									fb_ManipulatorArm( // Call Fb_Action
														(*Manipulator*)
															bCheckSensorManipulatorGripper:=GV_HMI.stTransferManipulatorToArm.bCheckSensorManipulatorGripper,
														(*Arm*)
															iGripperArmNumber:=GV_Cycle.iArmGripperLoad,
															bCheckSensorArmGripper1:=GV_HMI.stTransferManipulatorToArm.bCheckSensorArmGripper1,
															bCheckSensorArmGripper2:=GV_HMI.stTransferManipulatorToArm.bCheckSensorArmGripper2,
														(*Gripper*)
															tMouvementGripperOpen:=GV_HMI.stManipulatorGripper.tMouvementOpen,
															bCheckSensorGripperOpen:=GV_HMI.stManipulatorGripper.bCheckSensorOpen,
															tMouvementGripperClose:=GV_HMI.stManipulatorGripper.tMouvementClose,
															bCheckSensorGripperClose:=GV_HMI.stManipulatorGripper.bCheckSensorClose,
														(*Tunnel*)
															tTunnelTimeout:=GV_HMI.stManipulatorTunnel.tTimeout,
														(*Step 2_ManipulatorAboveTransfer*)
															tMove2Timeout:=T#0S, // Not used
														(*Step 3_ArmHome*)
															tMove3Timeout:=T#0S, // Not used
														(*Step 4_ManipulatorTransfer*)
															tMove4Timeout:=T#0S, // Not used
														(*Step 5_ArmTransfer*)
															tMove5Timeout:=T#0S, // Not used
														(*Step 7_ManipulatorAboveTransfer*)
															tMove7Timeout:=T#0S, // Not used
													 );
									IF fb_ManipulatorArm.bDone AND (NOT fb_ManipulatorArm.bError) THEN // Done 
										fb_ManipulatorArm.bStart:=FALSE; 
										GV_Cycle.bActionRunning:=FALSE;
										GV_Cycle.iSeqIndex:=GV_Cycle.iSeqIndex+1; 
									ELSIF fb_ManipulatorArm.bError THEN // Error
										fb_ManipulatorArm.bStart:=FALSE; 
										GV_Cycle.bActionRunning:=FALSE;
										GV_Cycle.udiErrorID:=2000+fb_ManipulatorArm.udiErrorID;
										GV_Cycle.bActionError:=TRUE;
									END_IF
									
								ENUM_Cycle_Action.ArmCNC:
								
									IF (NOT fb_ArmCNC.bInit) AND (NOT GV_Cycle.bActionRunning) THEN // Start if not already running	
										fb_ArmCNC.bStart:=TRUE;
										GV_Cycle.bActionRunning:=TRUE;
									END_IF
									
									IF fb_ArmCNC.bBusy THEN
										fb_ArmCNC.bStart:=FALSE;
									END_IF
									
									fb_ArmCNC( // Call Fb_Action
												(*TransferArmCnc*)
													bTransferArmToCnc:=GV_Cycle.bTransferArmToCnc,
													iGripperArmToCncNumber:=GV_Cycle.iGripperArmToCncNumber,
												(*TransferCncArm*)
													bTransferCncToArm:=GV_Cycle.bTransferCncToArm,
													iGripperCncToArmNumber:=GV_Cycle.iGripperCncToArmNumber,
												(*Arm*)
													bCheckSensorArmGripper1:=GV_HMI.stTransferArmCnc.bCheckSensorArmGripper1,
													bCheckSensorArmGripper2:=GV_HMI.stTransferArmCnc.bCheckSensorArmGripper2,
												(*Step 1_OpenDoor*)
													tMove1Timeout:=T#0S, // Not used
												(*Step 2_ArmInCNC*)
													tMove2Timeout:=T#0S, // Not used
												(*Step 3_WaitTransfer*)
													tMove3Timeout:=T#0S, // Not used
												(*Step 4_ArmHome*)
													tMove4Timeout:=T#0S, // Not used
												(*Step 5_CloseDoor*)
													tMove5Timeout:=T#0S, // Not used
											 );
									IF fb_ArmCNC.bDone AND (NOT fb_ArmCNC.bError) THEN // Done 
										fb_ArmCNC.bStart:=FALSE;
										GV_Cycle.bActionRunning:=FALSE; 
										GV_Cycle.iSeqIndex:=GV_Cycle.iSeqIndex+1; 
									ELSIF fb_ArmCNC.bError THEN // Error
										fb_ArmCNC.bStart:=FALSE;
										GV_Cycle.bActionRunning:=FALSE; 
										GV_Cycle.udiErrorID:=3000+fb_ArmCNC.udiErrorID;
										GV_Cycle.bActionError:=TRUE;
									END_IF
									
								ENUM_Cycle_Action.ArmToManipulator:
								
									IF (NOT fb_ArmManipulator.bInit) AND (NOT GV_Cycle.bActionRunning) THEN// Start if not already running	
										fb_ArmManipulator.bStart:=TRUE;
										GV_Cycle.bActionRunning:=TRUE;
									END_IF
									
									IF fb_ArmManipulator.bBusy THEN
										fb_ArmManipulator.bStart:=FALSE;
									END_IF
									
									fb_ArmManipulator( // Call Fb_Action
														(*Manipulator*)
															bCheckSensorManipulatorGripper:=GV_HMI.stTransferManipulatorToArm.bCheckSensorManipulatorGripper,
														(*Arm*)
															iGripperArmNumber:=GV_Cycle.iArmGripperUnload,
															bCheckSensorArmGripper1:=GV_HMI.stTransferArmToManipulator.bCheckSensorArmGripper1,
															bCheckSensorArmGripper2:=GV_HMI.stTransferArmToManipulator.bCheckSensorArmGripper2,
														(*Gripper*)
															tMouvementGripperOpen:=GV_HMI.stManipulatorGripper.tMouvementOpen,
															bCheckSensorGripperOpen:=GV_HMI.stManipulatorGripper.bCheckSensorOpen,
															tMouvementGripperClose:=GV_HMI.stManipulatorGripper.tMouvementClose,
															bCheckSensorGripperClose:=GV_HMI.stManipulatorGripper.bCheckSensorClose,
														(*Tunnel*)
															tTunnelTimeout:=GV_HMI.stManipulatorTunnel.tTimeout,
														(*Step 2_ManipulatorAboveTransfer*)
															tMove2Timeout:=T#0S, // Not used
														(*Step 3_ArmTransfer*)
															tMove3Timeout:=T#0S, // Not used
														(*Step 5_ManipulatorTransfer*)
															tMove5Timeout:=T#0S, // Not used
														(*Step 7_ArmHome*)
															tMove7Timeout:=T#0S, // Not used
														(*Step 8_ManipulatorAboveTransfer*)
															tMove8Timeout:=T#0S, // Not used
													);
									IF fb_ArmManipulator.bDone AND (NOT fb_ArmManipulator.bError) THEN // Done 
										fb_ArmManipulator.bStart:=FALSE; 
										GV_Cycle.bActionRunning:=FALSE;
										GV_Cycle.iSeqIndex:=GV_Cycle.iSeqIndex+1; 
									ELSIF fb_ArmManipulator.bError THEN // Error
										fb_ArmManipulator.bStart:=FALSE; 
										GV_Cycle.bActionRunning:=FALSE;
										GV_Cycle.udiErrorID:=4000+fb_ArmManipulator.udiErrorID;
										GV_Cycle.bActionError:=TRUE;
									END_IF
									
								ENUM_Cycle_Action.PlaceToolMagazine:
								
									IF GV_Cycle.iToolToUnloadLocationAbs=0 AND GV_Tool_Magazine.stManipulator.bToolPresenceMemory AND GV_Tool_Magazine.stManipulator.iAbsLocationNumberMemory<>GV_Cycle.iToolToLoadLocationAbs AND (NOT fb_PlaceToolMagazine.bStart) AND (NOT fb_PlaceToolMagazine.bInit) AND (NOT fb_PlaceToolMagazine.bBusy) THEN
										GV_Cycle.iToolToUnloadLocationAbs:=GV_Tool_Magazine.stManipulator.iAbsLocationNumberMemory;
									END_IF

									IF GV_Cycle.iToolToUnloadLocationAbs>0 THEN	
										//ICI -> Vérifier que emplacement disponible ? mémoire emplacement ou faire la vérif, avec outil en pince possible ?

										IF (NOT fb_PlaceToolMagazine.bInit) AND (NOT GV_Cycle.bActionRunning) THEN // Start if not already running		
											fb_PlaceToolMagazine.bStart:=TRUE;
											GV_Cycle.bActionRunning:=TRUE;
										END_IF
										
										IF fb_PlaceToolMagazine.bBusy THEN
											fb_PlaceToolMagazine.bStart:=FALSE;
										END_IF
										
										fb_PlaceToolMagazine( // Call Fb_Action
															(*ToolLocation*)
																stToolLocation:=GV_Tool_Magazine.aLocation[GV_Cycle.iToolToUnloadLocationAbs],
																lrZToolOffset:=GV_Tool_Magazine.lrZOffsetAboveLocation,//17.5,
															(*Manipulator*)
																bCheckSensorManipulatorGripper:=GV_HMI.stPickToolMagazine.bCheckSensorManipulatorGripper,
															(*Gripper*)
																tMouvementGripperOpen:=GV_HMI.stManipulatorGripper.tMouvementOpen,
																bCheckSensorGripperOpen:=GV_HMI.stManipulatorGripper.bCheckSensorOpen,
																tMouvementGripperClose:=GV_HMI.stManipulatorGripper.tMouvementClose,
																bCheckSensorGripperClose:=GV_HMI.stManipulatorGripper.bCheckSensorClose,
															(*Tunnel*)
																tTunnelTimeout:=GV_HMI.stManipulatorTunnel.tTimeout,
															(*Breakage*)
																tBreakageTimeout:=GV_HMI.stManipulatorBreakage.tTimeout,
																lrBreakageZOffsetSensor:=GV_HMI.stManipulatorBreakage.lrOffsetSensor,
																lrBreakageToleranceLength:=GV_HMI.stManipulatorBreakage.lrToleranceLength,
																lrBreakageVelocity:=GV_HMI.stManipulatorBreakage.lrMeasureVelocity,
															(*Step 4_FrontLocation*)
																tMove4Timeout:=T#0S, // Not used
															(*Step 6_AboveLocation*)
																tMove6Timeout:=T#0S, // Not used
															(*Step 8_FrontLocation*)
																tMove8Timeout:=T#0S, // Not used
															);
										IF fb_PlaceToolMagazine.bDone AND (NOT fb_PlaceToolMagazine.bError) THEN // Done 
											fb_PlaceToolMagazine.bStart:=FALSE; 
											GV_Cycle.bActionRunning:=FALSE;
											GV_Cycle.iToolToUnloadLocationAbs:=0;
											GV_Cycle.iSeqIndex:=GV_Cycle.iSeqIndex+1; 
										ELSIF fb_PlaceToolMagazine.bError THEN // Error
											GV_Cycle.udiErrorID:=5000+fb_PlaceToolMagazine.udiErrorID;
											GV_Cycle.bActionError:=TRUE;
										END_IF
										
									ELSE
										GV_Cycle.iSeqIndex:=GV_Cycle.iSeqIndex+1;
									END_IF
	
							END_CASE
							
						(* Action Error *)
							IF GV_Cycle.bActionError THEN // Action in Error
								(*Log*)
									PRG_Log_WM.fbLogWM.M_Write_Log('Cycle Step : 5_ExecuteSequence=Error');
									PRG_Log_WM.fbLogWM.M_Write_Log(CONCAT('Cycle Step : ErrorID=',UDINT_TO_STRING(GV_Cycle.udiErrorID)));
								GV_Cycle.eCycleStep:=ENUM_Cycle_Step.Error; // Go to Step Error
							END_IF		
				
					ELSE
						bExecuteSequenceDone:=TRUE;
					END_IF
					
				(* Next Step *)	
					IF bExecuteSequenceDone THEN
						GV_Cycle.eCycleStep:=ENUM_Cycle_Step.End; // Go to Step End
					END_IF
				
			ENUM_Cycle_Step.End: // Step End = 7
				bEndDone:=FALSE;
				GV_Cycle.iToolToUnloadLocationAbs:=0;
				(* End *)
					// ...
					IF ((GV_Cycle.bStartStop AND GV_Axes.bAxisAllNotMoving)
					OR ((NOT GV_Cycle.bStartStop) AND GV_Axes.stAxisX.bHaltDone AND GV_Axes.stAxisY.bHaltDone AND GV_Axes.stAxisZ.bHaltDone AND GV_Axes.stAxisArm.bHaltDone AND GV_Axes.bAxisAllNotMoving)) THEN
						GV_Axes.stAxisX.bAutoCmdAbs:=FALSE;
						GV_Axes.stAxisY.bAutoCmdAbs:=FALSE;
						GV_Axes.stAxisZ.bAutoCmdAbs:=FALSE;
						GV_Axes.stAxisArm.bAutoCmdAbs:=FALSE;
						bEndDone:=TRUE;
					END_IF

					//IF ((NOT GV_Cycle.bStartStop) AND GV_Axes.stAxisX.bStopDone AND GV_Axes.stAxisY.bStopDone AND GV_Axes.stAxisZ.bStopDone AND GV_Axes.stAxisArm.bStopDone AND GV_Axes.bAxisAllNotMoving) THEN
					//	bEndDone:=TRUE;
					//END_IF
					
				(* Next Step *)	
					IF bEndDone THEN
						GV_Cycle.eCycleStep:=ENUM_Cycle_Step.InitData; // Go to Step InitData
					END_IF
	
			ENUM_Cycle_Step.Error: // Step Error = 9
				bErrorDone:=FALSE;
				GV_Cycle.iToolToUnloadLocationAbs:=0;
				(* Error *)
					// ...
					GV_Axes.stAxisX.bAutoCmdAbs:=FALSE;
					GV_Axes.stAxisY.bAutoCmdAbs:=FALSE;
					GV_Axes.stAxisZ.bAutoCmdAbs:=FALSE;
					GV_Axes.stAxisArm.bAutoCmdAbs:=FALSE;
					
					GV_Cycle.bStartStop:=FALSE;
					GV_Cycle.bInitCycleDone:=FALSE;
					
					IF GV_Cycle.bResetError THEN
						bErrorDone:=TRUE;
					END_IF
				(* Next Step *)	
					IF bErrorDone THEN
						GV_Cycle.bActionRunning:=FALSE;
						GV_Cycle.bActionError:=FALSE;
						GV_Cycle.udiErrorID:=0;
						GV_Cycle.eCycleStep:=ENUM_Cycle_Step.InitData;
					END_IF
			
		END_CASE
		
	END_IF

(** CYCLE IN PROGRESS **)
GV_Cycle.bCycleInProgress:=GV_Cycle.eCycleStep<>ENUM_Cycle_Step.InitAll AND GV_Cycle.eCycleStep<>ENUM_Cycle_Step.InitData;

(** LOG CYCLE STEP **)
	(* Text CycleStep *)
		CASE GV_Cycle.eCycleStep OF
				ENUM_Cycle_Step.InitAll:           	sTxtCycleStep:='0_InitAll';
				ENUM_Cycle_Step.InitData:           sTxtCycleStep:='0_InitData';
				ENUM_Cycle_Step.Ready:          	sTxtCycleStep:='2_Ready';
				ENUM_Cycle_Step.Preparation:        sTxtCycleStep:='3_Preparation';
				ENUM_Cycle_Step.BuildSequence:  	sTxtCycleStep:='4_BuildSequence';
				ENUM_Cycle_Step.ExecuteSequence:	sTxtCycleStep:='5_ExecuteSequence';
				ENUM_Cycle_Step.End:            	sTxtCycleStep:='7_End';
				ENUM_Cycle_Step.Abort:          	sTxtCycleStep:='8_Abort';
				ENUM_Cycle_Step.Error:         		sTxtCycleStep:='9_Error';
		END_CASE
	(* Text CyclePrevStep *)
		CASE GV_Cycle.eCyclePrevStep OF
				ENUM_Cycle_Step.InitAll:           	sTxtCycleStep:='0_InitAll';
				ENUM_Cycle_Step.InitData:           sTxtCycleStep:='0_InitData';
				ENUM_Cycle_Step.Ready:          	sTxtCycleStep:='2_Ready';
				ENUM_Cycle_Step.Preparation:        sTxtCycleStep:='3_Preparation';
				ENUM_Cycle_Step.BuildSequence:  	sTxtCycleStep:='4_BuildSequence';
				ENUM_Cycle_Step.ExecuteSequence:	sTxtCycleStep:='5_ExecuteSequence';
				ENUM_Cycle_Step.End:            	sTxtCycleStep:='7_End';
				ENUM_Cycle_Step.Abort:          	sTxtCycleStep:='8_Abort';
				ENUM_Cycle_Step.Error:         		sTxtCycleStep:='9_Error';
		END_CASE
	(* Log *)
		sTextLog:=(CONCAT('Cycle Step ',CONCAT(sTxtCyclePrevStep,CONCAT('-> ',sTxtCycleStep))));	
		IF GV_OpMode.eOpMode=ENUM_OpMode.AUTO AND GV_Cycle.eCycleStep<>GV_Cycle.eCyclePrevStep THEN
			PRG_Log_WM.fbLogWM.M_Write_Log(sTextLog);
			GV_Cycle.eCyclePrevStep:=GV_Cycle.eCycleStep; // Previous Step := Step in progress
		END_IF

END_PROGRAM

// ---- 08_Cycle/03_POUs/02_FBs/FB_20_Action_Initialization.TcPOU
FUNCTION_BLOCK FB_20_Action_Initialization
VAR_INPUT
	(** SETUP ST **)
		//stToolLocation : ST_Tool_Location ; // Tool_Location structure of the Tool to Pick
		
	(** SETUP TIME **)
		(*Manipulator Gripper mvmnt*)
			//tMouvementGripperOpen : TIME ; // Value of the manipulator gripper open mouvement duration
			//tMouvementGripperClose : TIME ; // Value of the manipulator gripper close mouvement duration
		(*Tunnel*)
			tTunnelTimeout : TIME ; // Value of the timeout for travel the tunnel
		(*Step 2*)
			tMove2Timeout : TIME ; // Value of the timeout for Step 2

	(** SETUP FLAG **)
		//bCheckSensorManipulatorGripper : BOOL ; // Check the manipulator gripper sensor at the beginning
		(*Gripper*)
			//bCheckSensorGripperOpen : BOOL ; // Check the manipulator gripper sensor after open
			//bCheckSensorGripperClose : BOOL ; // Check the manipulator gripper sensor after close	
			
	(** PROCESS FLAG **)
	    bInit : BOOL ; // Init the Fb
	    bStart : BOOL ; // Start the Fb
END_VAR
VAR_OUTPUT
	(** PROCESS UDINT **)
		udiErrorID : UDINT ; // Fb Error ID
		
	(** PROCESS FLAG **)
		bBusy  : BOOL ; // Fb is Busy
		bDone  : BOOL ; // Fb is Done
		bError : BOOL ; // Fb in Error
END_VAR
VAR_IN_OUT
END_VAR	
VAR
	(** SETUP ENUM **)
		(*Manipulator Gripper mvmnt*)
			//eGripperMode : ENUM_Gripper_Mode; // Gripper mode for gripper mouvement (fbGripper)
		(*Tunnel*)
			eTunnelMode : ENUM_Tunnel_Mode; // Tunnel mode for travel (fbTunnel)

	(** SETUP TIME **)
		(*Manipulator Gripper mvmnt*)
			//tGripperTime : TIME ; // Mouvement duration for gripper mouvement (fbGripper)
	
	(** SETUP FLAG **)
		(*Manipulator Gripper mvmnt*)
			//bGripperSensor : BOOL ; // Sensor check for gripper mouvement (fbGripper)
		
	(** PROCESS STRING **)
		strTextLog : STRING ; // Text to Log
		
	(** PROCESS LREAL **)
		
	(** PROCESS INT **)
		iStep  : INT := 0 ; // Step of the Fb
		iSubStep : INT := 0 ; // SubStep of the Fb
		iPrevStep : INT := 0 ; // Previous Step of the Fb
		iPrevSubStep : INT := 0 ; // Previous Subtep of the Fb
		
	(** PROCESS FLAG + R_TRIG **)
		rtInit : R_TRIG ; // FB Init at rising edge
		rtStart : R_TRIG ; // FB Start at rising edge
		(*Tunnel*)
			bTunnelTravel : BOOL ; // Need to travel the tunnel
		bXError : BOOL ; // Axis X Error
		bYError : BOOL ; // Axis Y Error
		bZError : BOOL ; // Axis Z Error
		bArmError : BOOL ; // Axis Arm Error
	
	(** FB **)
		(*Gripper*)
			//fbGripper : FB_Manipulator_Gripper ;
		(*Tunnel*)
			fbTunnel : FB_Manipulator_Tunnel ;
		(*Step 2*)
			tonTimeoutMove2 : TON ; // TON timeout for the Step 2
END_VAR

//-----------------------------------------------------------------------------------------
//
//                  			FB_20_Action_Initialization
//
//						Management of the Initialization process
//-----------------------------------------------------------------------------------------
//
//Auteur: G.GOETZ
//Création: 13.03.2026
//Dernière modification : 13.03.2026 (G.GOETZ)
//       			
//-----------------------------------------------------------------------------------------
//
//     							Liste des modifications  	
//
// 13.03.2026 (G.GOETZ) -> Création		
//-----------------------------------------------------------------------------------------

(** FB CALL **)
	rtInit(CLK:=bInit);
	rtStart(CLK:=bStart);
	fbTunnel( // Call Tunnel travel
			eTunnelMode:=eTunnelMode,
			tTimeout:=tTunnelTimeout
			);

(** AXIS ERRORS **)
	bXError:=(GV_Axes.stAxisX.stDriveAx8206.AxisRef.Status.Error OR GV_Axes.stAxisX.stDriveAx8206.AxisRef.Status.ErrorStop OR GV_Axes.stAxisX.stDriveAx8206.AxisRef.Status.ErrorID<>0);
	bYError:=(GV_Axes.stAxisY.stDriveAx8206.AxisRef.Status.Error OR GV_Axes.stAxisY.stDriveAx8206.AxisRef.Status.ErrorStop OR GV_Axes.stAxisY.stDriveAx8206.AxisRef.Status.ErrorID<>0);
	bZError:=(GV_Axes.stAxisZ.stDriveAx8206.AxisRef.Status.Error OR GV_Axes.stAxisZ.stDriveAx8206.AxisRef.Status.ErrorStop OR GV_Axes.stAxisZ.stDriveAx8206.AxisRef.Status.ErrorID<>0);
	bArmError:=(GV_Axes.stAxisArm.stDriveAx8206.AxisRef.Status.Error OR GV_Axes.stAxisArm.stDriveAx8206.AxisRef.Status.ErrorStop OR GV_Axes.stAxisArm.stDriveAx8206.AxisRef.Status.ErrorID<>0);


(** INIT **)
	IF (rtinit.Q OR bInit) AND (NOT bStart) THEN
		bBusy:=FALSE;
		bDone:=FALSE;
		bError:=FALSE;
		udiErrorID:=0;
		iStep:=0;
		iSubStep:=0;
		bInit:=FALSE;
	END_IF

(** STEPS **)
    CASE iStep OF
		
        0: (* Step 0 = Idle + Check *)
            bBusy:=FALSE;
            bDone:=FALSE;
			bError:=FALSE;
			udiErrorID:=0;
			iSubStep:=0;
			
			tonTimeoutMove2.IN:=FALSE;
			//tonTimeoutMove4.IN:=FALSE;
			//tonTimeoutMove6.IN:=FALSE;
			//tonTimeoutMove8.IN:=FALSE;
			
			GV_Axes.stAxisX.bAutoCmdAbs:=FALSE;
			GV_Axes.stAxisY.bAutoCmdAbs:=FALSE;
			GV_Axes.stAxisZ.bAutoCmdAbs:=FALSE;
			GV_Axes.stAxisArm.bAutoCmdAbs:=FALSE;
			
			fbTunnel.bInit:=TRUE;
			
			bTunnelTravel:=FALSE;

			(* Idle->Start *)
				IF rtStart.Q AND (NOT bInit) THEN
					bBusy:=TRUE;
					(*Log*)
						PRG_Log_WM.fbLogWM.M_Write_Log('FB_20_Action_Initialization : 0_Idle : Init of the Magazine');
						//IF Exemple THEN
						//	strTextLog:='With';
						//ELSE
						//	strTextLog:='Without';
						//END_IF
						//PRG_Log_WM.fbLogWM.M_Write_Log(CONCAT('FB_20_Action_Initialization : 0_Idle : Exemple Check = ',strTextLog));
							
					(* Check xxx *)

					IF (NOT bError) THEN
						(*Log*)
							PRG_Log_WM.fbLogWM.M_Write_Log('FB_20_Action_Initialization : 0_Idle->1_Tunnel');
						iStep:=1; // Next Step
					END_IF

				END_IF
	
		1: (* Step 1 = Tunnel passage (if needed) *)
			IF (NOT bTunnelTravel) THEN
				IF GV_Tool_Magazine.stManipulator.ePositionMag=ENUM_Position_Magazine.Top THEN
					bTunnelTravel:=FALSE;
					(*Log*)
						PRG_Log_WM.fbLogWM.M_Write_Log('FB_20_Action_Initialization : 1_Tunnel : No Need to Travel');
						PRG_Log_WM.fbLogWM.M_Write_Log('FB_20_Action_Initialization : 1_Tunnel->2_???');
					iStep:=2; // Next Step
				END_IF	
				IF GV_Tool_Magazine.stManipulator.ePositionMag=ENUM_Position_Magazine.Bottom THEN
					eTunnelMode:=ENUM_Tunnel_MODE.BottomToTop;
					bTunnelTravel:=TRUE;
					(*Log*)
						PRG_Log_WM.fbLogWM.M_Write_Log('FB_20_Action_Initialization : 1_Tunnel : Need to Travel Bottom->Top');
				END_IF			
				IF GV_Tool_Magazine.stManipulator.ePositionMag=ENUM_Position_Magazine.Unknow THEN // Manipulator Unknow position
					bError:=TRUE;
					udiErrorID:=101; // 101 = Step 1 Error Tunnel 01
					fbTunnel.bStart:=FALSE;
					bTunnelTravel:=FALSE;
					(*Log*)
						PRG_Log_WM.fbLogWM.M_Write_Log('FB_20_Action_Initialization : 1_Tunnel=Error');
						PRG_Log_WM.fbLogWM.M_Write_Log(CONCAT('FB_20_Action_Initialization : ErrorID=',UDINT_TO_STRING(udiErrorID)));
					iStep:=0; // Idle Step
				END_IF
			END_IF
			
			IF bTunnelTravel AND (NOT fbTunnel.bStart) AND (NOT fbTunnel.bBusy) THEN // Tunnel Start
				fbTunnel.bStart:=TRUE;
			END_IF
			IF fbTunnel.bDone THEN // Tunnel Done
				fbTunnel.bStart:=FALSE;
				bTunnelTravel:=FALSE;
				(*Log*)
					PRG_Log_WM.fbLogWM.M_Write_Log('FB_20_Action_Initialization : 1_Tunnel->2_???');
				iStep:=2; // Next Step
			ELSIF fbTunnel.bError THEN // Tunnel Error
				bError:=TRUE;
				udiErrorID:=100+fbTunnel.udiErrorID; // 1xx = Step 1 Error + Error xx fbTunnel
				fbTunnel.bStart:=FALSE;
				bTunnelTravel:=FALSE;
				(*Log*)
					PRG_Log_WM.fbLogWM.M_Write_Log('FB_20_Action_Initialization : 1_Tunnel=Error');
					PRG_Log_WM.fbLogWM.M_Write_Log(CONCAT('FB_20_Action_Initialization : ErrorID=',UDINT_TO_STRING(udiErrorID)));
				iStep:=0; // Idle Step
			END_IF
		
		2: (* Step 2 = Move the manipulator to Home (Y->Z->X) *)
			tonTimeoutMove2.PT:=tMove2Timeout;
			tonTimeoutMove2.IN:=TRUE;
			
			CASE iSubStep OF
        
				0: (* Start Y move *)
					GV_Axes.stAxisY.lrAutoPosAbs:=GV_Tool_Magazine.stManipulator.lrYHome;
					GV_Axes.stAxisY.bAutoCmdAbs:=TRUE;
					(*Log*)
						PRG_Log_WM.fbLogWM.M_Write_Log('FB_20_Action_Initialization : 2_MoveHome : 0 : Start Y move');
					iSubStep:=1; // Next SubStep

				1: (* Wait Y move done *)
				   IF GV_Axes.stAxisY.bAutoDone AND (NOT bYError) THEN
						GV_Axes.stAxisY.bAutoCmdAbs:=FALSE;
						(*Log*)
							PRG_Log_WM.fbLogWM.M_Write_Log('FB_20_Action_Initialization : 2_MoveHome : 1 : Y move done');
						iSubStep:=2; // Next SubStep
					ELSIF bYError THEN
						bError:=TRUE;
						udiErrorID:=211; // 211 = Step 2 SubStep 1 Error Axis Y 1
						GV_Axes.stAxisY.bAutoCmdAbs:=FALSE;
						tonTimeoutMove2.IN:=FALSE;
						(*Log*)
							PRG_Log_WM.fbLogWM.M_Write_Log('FB_20_Action_Initialization : 2_MoveHome=Error');
							PRG_Log_WM.fbLogWM.M_Write_Log(CONCAT('FB_20_Action_Initialization : ErrorID=',UDINT_TO_STRING(udiErrorID)));
						iSubStep:=0; // Stop SubStep
						iStep:=0; // Idle Step
					END_IF
				
				2: (* Start Z move *)
					GV_Axes.stAxisZ.lrAutoPosAbs:=GV_Tool_Magazine.stManipulator.lrZHome;
					GV_Axes.stAxisZ.bAutoCmdAbs:=TRUE;
					(*Log*)
						PRG_Log_WM.fbLogWM.M_Write_Log('FB_20_Action_Initialization : 2_MoveHome : 2 : Start Z move');
					iSubStep:=3; // Next SubStep

				3: (* Wait Z move done *)
				   IF GV_Axes.stAxisZ.bAutoDone AND (NOT bZError) THEN
						GV_Axes.stAxisZ.bAutoCmdAbs:=FALSE;
						(*Log*)
							PRG_Log_WM.fbLogWM.M_Write_Log('FB_20_Action_Initialization : 2_MoveHome : 3 : Z move done');
						iSubStep:=4; // Next SubStep
					ELSIF bZError THEN
						bError:=TRUE;
						udiErrorID:=231; // 231 = Step 2 SubStep 3 Error Axis Z 1
						GV_Axes.stAxisZ.bAutoCmdAbs:=FALSE;
						tonTimeoutMove2.IN:=FALSE;
						(*Log*)
							PRG_Log_WM.fbLogWM.M_Write_Log('FB_20_Action_Initialization : 2_MoveHome=Error');
							PRG_Log_WM.fbLogWM.M_Write_Log(CONCAT('FB_20_Action_Initialization : ErrorID=',UDINT_TO_STRING(udiErrorID)));
						iSubStep:=0; // Stop SubStep
						iStep:=0; // Idle Step
					END_IF

				4: (* Start X move *)
					GV_Axes.stAxisX.lrAutoPosAbs:=GV_Tool_Magazine.stManipulator.lrXHome;
					GV_Axes.stAxisX.bAutoCmdAbs:=TRUE;
					(*Log*)
						PRG_Log_WM.fbLogWM.M_Write_Log('FB_20_Action_Initialization : 2_MoveHome : 4 : Start X move');
					iSubStep:=5; // Next Step

				5: (* Wait X move done *)
				   IF GV_Axes.stAxisX.bAutoDone AND (NOT bXError) THEN
						GV_Axes.stAxisX.bAutoCmdAbs:=FALSE;
						tonTimeoutMove2.IN:=FALSE;
						(*Log*)
							PRG_Log_WM.fbLogWM.M_Write_Log('FB_20_Action_Initialization : 2_MoveHome : 5 : X move done');
							PRG_Log_WM.fbLogWM.M_Write_Log('FB_20_Action_Initialization : 2_MoveHome->0_Idle');
						iSubStep:=0; // End SubStep
						iStep:=0; // End Step
						bDone:=TRUE;
						bBusy:=FALSE;
					ELSIF bXError THEN
						bError:=TRUE;
						udiErrorID:=251; // 251 = Step 2 SubStep 5 Error Axis X 1
						GV_Axes.stAxisX.bAutoCmdAbs:=FALSE;
						tonTimeoutMove2.IN:=FALSE;
						(*Log*)
							PRG_Log_WM.fbLogWM.M_Write_Log('FB_20_Action_Initialization : 2_MoveHome=Error');
							PRG_Log_WM.fbLogWM.M_Write_Log(CONCAT('FB_20_Action_Initialization : ErrorID=',UDINT_TO_STRING(udiErrorID)));
						iSubStep:=0; // Stop SubStep
						iStep:=0; // Idle Step
					END_IF
					
			END_CASE	
		
			IF tonTimeoutMove2.Q AND tonTimeoutMove2.PT<>T#0S THEN // Timeout 
				bError:=TRUE;
				udiErrorID:=299; // 299 = Step 2 Error Timeout 99
				GV_Axes.stAxisZ.bAutoCmdAbs:=FALSE;
				GV_Axes.stAxisX.bAutoCmdAbs:=FALSE;
				GV_Axes.stAxisY.bAutoCmdAbs:=FALSE;
				tonTimeoutMove2.IN:=FALSE;
				(*Log*)
					PRG_Log_WM.fbLogWM.M_Write_Log('FB_20_Action_Initialization : 2_MoveHome=Error');
					PRG_Log_WM.fbLogWM.M_Write_Log(CONCAT('FB_20_Action_Initialization : ErrorID=',UDINT_TO_STRING(udiErrorID)));
				iSubStep:=0;
				iStep:=0;
			END_IF
			
			
			
			
	END_CASE

END_FUNCTION_BLOCK

// ---- 09_Tool_Magazine/03_POUs/02_FBs/FB_Manipulator_Tunnel.TcPOU
FUNCTION_BLOCK FB_Manipulator_Tunnel
VAR_INPUT
	(** SETUP ENUM **)
		eTunnelMode : ENUM_Tunnel_Mode ; // Mode of the tunnel	

	(** SETUP TIME **)
		tTimeout : TIME ; // Max time for travel the tunnel

	(** PROCESS FLAG **)
		bInit : BOOL ; // Init the FB
	    bStart : BOOL ; // Start the Fb
END_VAR
VAR_OUTPUT
	(** PROCESS UDINT **)
		udiErrorID : UDINT ; // Fb Error ID
		
	(** PROCESS FLAG **)
		bBusy  : BOOL ; // Fb is Busy
		bDone  : BOOL ; // Fb is Done
		bError : BOOL ; // Fb in Error
END_VAR
VAR_IN_OUT
END_VAR	
VAR
	(** STRING **)
		strTextLog : STRING ; // Text to Log

	(** PROCESS INT **)
		iStep  : INT := 0 ; // Step of the Fb
		iSubStep : INT := 0 ; // SubStep of the Fb
		iPrevStep : INT := 0 ; // Previous Step of the Fb
		iPrevSubStep : INT := 0 ; // Previous Subtep of the Fb
	
	(** PROCESS FLAG + R_TRIG **)
		rtInit : R_TRIG ; // FB Init at rising edge
		rtStart : R_TRIG ; // FB Start at rising edge
		bTunnelTravelDone : BOOL ; // Tunnel travel done
		bXError : BOOL ; // Axis X Error
		bYError : BOOL ; // Axis Y Error
		bZError : BOOL ; // Axis Z Error
		bArmError : BOOL ; // Axis Arm Error
		
	(** FB **)
		tonTimeout : TON ; // TON timeout of the tunnel travel
END_VAR

//-----------------------------------------------------------------------------------------
//
//                  		FB_Manipulator_Tunnel
//
//			Management of the manipulator passage through the tunnel
//-----------------------------------------------------------------------------------------
//
//Auteur: G.GOETZ
//Création: 06.02.2026
//Dernière modification : 08.04.2026 (G.GOETZ)
//       			
//-----------------------------------------------------------------------------------------
//
//     							Liste des modifications  	
//
// 06.02.2026 (G.GOETZ) -> Création
// 08.04.2026 (G.GOETZ) -> Ajout Init + Modification du cycle
//-----------------------------------------------------------------------------------------

(** FB CALL **)
	rtInit(CLK:=bInit);
	rtStart(CLK:=bStart);
	
	tonTimeout();

(** AXIS ERRORS **)
	bXError:=(GV_Axes.stAxisX.stDriveAx8206.AxisRef.Status.Error OR GV_Axes.stAxisX.stDriveAx8206.AxisRef.Status.ErrorStop OR GV_Axes.stAxisX.stDriveAx8206.AxisRef.Status.ErrorID<>0);
	bYError:=(GV_Axes.stAxisY.stDriveAx8206.AxisRef.Status.Error OR GV_Axes.stAxisY.stDriveAx8206.AxisRef.Status.ErrorStop OR GV_Axes.stAxisY.stDriveAx8206.AxisRef.Status.ErrorID<>0);
	bZError:=(GV_Axes.stAxisZ.stDriveAx8206.AxisRef.Status.Error OR GV_Axes.stAxisZ.stDriveAx8206.AxisRef.Status.ErrorStop OR GV_Axes.stAxisZ.stDriveAx8206.AxisRef.Status.ErrorID<>0);
	bArmError:=(GV_Axes.stAxisArm.stDriveAx8206.AxisRef.Status.Error OR GV_Axes.stAxisArm.stDriveAx8206.AxisRef.Status.ErrorStop OR GV_Axes.stAxisArm.stDriveAx8206.AxisRef.Status.ErrorID<>0);

(** INIT **)
	IF (rtinit.Q OR bInit) AND (NOT bStart) THEN
		iStep:=0;
		bInit:=FALSE;
	END_IF

(** STEPS **)
    CASE iStep OF
		
        0: (* Step 0 = Idle *)
            bBusy:=FALSE;
            bDone:=FALSE;
			bError:=FALSE;
			udiErrorID:=0;
			iSubStep:=0;
			
			tonTimeout.IN:=FALSE;
			
			bTunnelTravelDone:=FALSE;
			
			(* Idle->Setup *)
				IF bStart AND (NOT bInit) THEN
					bBusy:=TRUE;
					(*Log*)
						PRG_Log_WM.fbLogWM.M_Write_Log('FB_Manipulator_Tunnel : 0_Idle->1_Setup');
					iStep:=1; // Next Step
				END_IF
				
		1: (* Step 1 = Setup *)
			(*Log*)
				(*TunnelMode*)
					CASE eTunnelMode OF
						ENUM_Tunnel_Mode.TopToBottom:		strTextLog:='TopToBottom';
						ENUM_Tunnel_Mode.BottomToTop:		strTextLog:='BottomToTop';
					END_CASE
					PRG_Log_WM.fbLogWM.M_Write_Log(CONCAT('FB_Manipulator_Tunnel : 1_Setup : Tunnel Mode = ',strTextLog));
				(*Timeout*)
					strTextLog:=TIME_TO_STRING(tTimeout);
					PRG_Log_WM.fbLogWM.M_Write_Log(CONCAT('FB_Manipulator_Tunnel : 1_Setup : Timeout = ',strTextLog));				
				PRG_Log_WM.fbLogWM.M_Write_Log('FB_Manipulator_Tunnel : 1_Setup->2_Process');
				
			tonTimeout.PT:=tTimeout;
			iStep:=2; // Next Step
			
		2: (* Step 2 = Process (Y->(ZLowestRacKTop)->(XFirst)) *)
			tonTimeout.IN:=TRUE; // Start TON timeout

				CASE iSubStep OF
		
					0: (* Start Y move *)
						GV_Axes.stAxisY.lrAutoPosAbs:=GV_Tool_Magazine.stManipulator.lrYTunnel;
						GV_Axes.stAxisY.bAutoCmdAbs:=TRUE;
						(*Log*)
							PRG_Log_WM.fbLogWM.M_Write_Log('FB_Manipulator_Tunnel : 2_Process : 0 : Start Y move');
						iSubStep:=1; // Next SubStep
						
					1: (* Wait Y move done *)
					   IF GV_Axes.stAxisY.bAutoDone AND (NOT bYError) THEN
							GV_Axes.stAxisY.bAutoCmdAbs:=FALSE;
							(*Log*)
								PRG_Log_WM.fbLogWM.M_Write_Log('FB_Manipulator_Tunnel : 2_Process : 1 : Y move done');

							CASE eTunnelMode OF 
								ENUM_Tunnel_Mode.TopToBottom: // X Top
									IF GV_Tool_Magazine.stManipulator.lrZPosition<GV_Tool_Magazine.lrZLowestRackTop+40 THEN
										(*Log*)
											PRG_Log_WM.fbLogWM.M_Write_Log('FB_Manipulator_Tunnel : 2_Process : 1->2 : ZLowestRackTop');
										iSubStep:=2; // Next SubStep
									ELSE
										IF GV_Tool_Magazine.stManipulator.lrXPosition<GV_Tool_Magazine.lrXFirstLocationTop THEN
											(*Log*)
												PRG_Log_WM.fbLogWM.M_Write_Log('FB_Manipulator_Tunnel : 2_Process : 1->4 : XFirstTop');
											iSubStep:=4; // Next SubStep
										ELSE
											(*Log*)
												PRG_Log_WM.fbLogWM.M_Write_Log('FB_Manipulator_Tunnel : 2_Process -> 3_Process');
											iSubStep:=0; // End SubStep
											iStep:=3; // Next Stpe
										END_IF
									END_IF
								ENUM_Tunnel_Mode.BottomToTop: // X Bottom
									IF GV_Tool_Magazine.stManipulator.lrXPosition<GV_Tool_Magazine.lrXFirstLocationBottom+GV_Tool_Magazine.lrXLocationOffsetBottom THEN
										(*Log*)
											PRG_Log_WM.fbLogWM.M_Write_Log('FB_Manipulator_Tunnel : 2_Process : 1->4 : XFirstBottom');
										iSubStep:=4; // Next SubStep
									ELSE
										(*Log*)
											PRG_Log_WM.fbLogWM.M_Write_Log('FB_Manipulator_Tunnel : 2_Process -> 3_Process');
											iSubStep:=0; // End SubStep
											iStep:=3; // Next Stpe
									END_IF
							END_CASE
						ELSIF bYError THEN
							bError:=TRUE;
							udiErrorID:=21; // 21 = Step 2 SubStep 1 Error Axis Y
							GV_Axes.stAxisY.bAutoCmdAbs:=FALSE;
							tonTimeout.IN:=FALSE;
							(*Log*)
								PRG_Log_WM.fbLogWM.M_Write_Log('FB_Manipulator_Tunnel : 2_Process=Error');
								PRG_Log_WM.fbLogWM.M_Write_Log(CONCAT('FB_Manipulator_Tunnel : ErrorID=',UDINT_TO_STRING(udiErrorID)));
							iSubStep:=0; // Stop SubStep
							iStep:=0; // Idle Step
						END_IF

					2: (* Start ZLowestRackTop move *)
						GV_Axes.stAxisZ.lrAutoPosAbs:=GV_Tool_Magazine.lrZLowestRackTop+40;
						(*Log*)
							PRG_Log_WM.fbLogWM.M_Write_Log('FB_Manipulator_Tunnel : 2_Process : 2 : Start ZLowestRackTop move');
						GV_Axes.stAxisZ.bAutoCmdAbs:=TRUE;
						iSubStep:=3; // Next SubStep

					3: (* Wait ZLowestRackTop move done *)
					   IF GV_Axes.stAxisZ.bAutoDone AND (NOT bZError) THEN
							GV_Axes.stAxisZ.bAutoCmdAbs:=FALSE;
							(*Log*)
								PRG_Log_WM.fbLogWM.M_Write_Log('FB_Manipulator_Tunnel : 2_Process : 3 : ZLowestRackTop move done');
							iSubStep:=0; // End SubStep
							iStep:=4; // Next STep
						ELSIF bZError THEN
							bError:=TRUE;
							udiErrorID:=23; // 23 = Step 2 SubStep 3 Error Axis Z
							GV_Axes.stAxisZ.bAutoCmdAbs:=FALSE;
							tonTimeout.IN:=FALSE;
							(*Log*)
								PRG_Log_WM.fbLogWM.M_Write_Log('FB_Manipulator_Tunnel : 2_Process=Error');
								PRG_Log_WM.fbLogWM.M_Write_Log(CONCAT('FB_Manipulator_Tunnel : ErrorID=',UDINT_TO_STRING(udiErrorID)));
							iSubStep:=0; // Stop 
							iStep:=0; // Idle Step
						END_IF
						
					4: (* Start XFirst move *)
						CASE eTunnelMode OF 
							ENUM_Tunnel_Mode.TopToBottom: // X Top
								GV_Axes.stAxisX.lrAutoPosAbs:=GV_Tool_Magazine.lrXFirstLocationTop;
								(*Log*)
									PRG_Log_WM.fbLogWM.M_Write_Log('FB_Manipulator_Tunnel : 2_Process : 4 : Start XFirstTop move');
							ENUM_Tunnel_Mode.BottomToTop: // X Bottom
								GV_Axes.stAxisX.lrAutoPosAbs:=GV_Tool_Magazine.lrXFirstLocationBottom+GV_Tool_Magazine.lrXLocationOffsetBottom;
								(*Log*)
									PRG_Log_WM.fbLogWM.M_Write_Log('FB_Manipulator_Tunnel : 2_Process : 4 : Start XFirstBottom move');
						END_CASE
						GV_Axes.stAxisX.bAutoCmdAbs:=TRUE;
						iSubStep:=5; // Next SubStep

					5: (* Wait XFirst move done *)
					   IF GV_Axes.stAxisX.bAutoDone AND (NOT bXError) THEN
							GV_Axes.stAxisX.bAutoCmdAbs:=FALSE;
							(*Log*)
								PRG_Log_WM.fbLogWM.M_Write_Log('FB_Manipulator_Tunnel : 2_Process : 5 : XFirst move done');
							iSubStep:=0; // End SubStep
							iStep:=3; // Next STep
						ELSIF bXError THEN
							bError:=TRUE;
							udiErrorID:=25; // 25 = Step 2 SubStep 5 Error Axis X
							GV_Axes.stAxisX.bAutoCmdAbs:=FALSE;
							tonTimeout.IN:=FALSE;
							(*Log*)
								PRG_Log_WM.fbLogWM.M_Write_Log('FB_Manipulator_Tunnel : 2_Process=Error');
								PRG_Log_WM.fbLogWM.M_Write_Log(CONCAT('FB_Manipulator_Tunnel : ErrorID=',UDINT_TO_STRING(udiErrorID)));
							iSubStep:=0; // Stop 
							iStep:=0; // Idle Step
						END_IF
						
				END_CASE
				
			IF tonTimeout.Q AND tonTimeout.PT<>T#0S THEN
				bError:=TRUE;
				udiErrorID:=29; // 29 = Step 2 Error Timeout 9
				GV_Axes.stAxisZ.bAutoCmdAbs:=FALSE;
				GV_Axes.stAxisX.bAutoCmdAbs:=FALSE;
				GV_Axes.stAxisY.bAutoCmdAbs:=FALSE;
				tonTimeout.IN:=FALSE;
				(*Log*)
					PRG_Log_WM.fbLogWM.M_Write_Log('FB_Manipulator_Tunnel : 2_Process : Error');
					PRG_Log_WM.fbLogWM.M_Write_Log(CONCAT('FB_Manipulator_Tunnel : ErrorID = ',UDINT_TO_STRING(udiErrorID)));
				iSubStep:=0; // Stop SubStep
				iStep:=0; // Idle Step
			END_IF
			
		3: (* Step 3 = Process (X->Z) *)	
				CASE iSubStep OF

					0: (* Start X move *)
						GV_Axes.stAxisX.lrAutoPosAbs:=GV_Tool_Magazine.stManipulator.lrXTunnel;
						GV_Axes.stAxisX.bAutoCmdAbs:=TRUE;
						(*Log*)
							PRG_Log_WM.fbLogWM.M_Write_Log('FB_Manipulator_Tunnel : 3_Process : 0 : Start X move');
						iSubStep:=1; // Next SubStep
		
					1: (* Wait X move done *)
					   IF GV_Axes.stAxisX.bAutoDone AND (NOT bXError) THEN
							GV_Axes.stAxisX.bAutoCmdAbs:=FALSE;
							(*Log*)
								PRG_Log_WM.fbLogWM.M_Write_Log('FB_Manipulator_Tunnel : 3_Process : 1 : X move done');
							iSubStep:=2; // Next SubStep
						ELSIF bXError THEN
							bError:=TRUE;
							udiErrorID:=31; // 31 = Step 3 SubStep 1 Error Axis X
							GV_Axes.stAxisX.bAutoCmdAbs:=FALSE;
							tonTimeout.IN:=FALSE;
							(*Log*)
								PRG_Log_WM.fbLogWM.M_Write_Log('FB_Manipulator_Tunnel : 3_Process=Error');
								PRG_Log_WM.fbLogWM.M_Write_Log(CONCAT('FB_Manipulator_Tunnel : ErrorID=',UDINT_TO_STRING(udiErrorID)));
							iSubStep:=0; // Stop SubStep
							iStep:=0; // Idle Step
						END_IF

					2: (* Start Z move *)
						CASE eTunnelMode OF 
							ENUM_Tunnel_Mode.TopToBottom: // Z bottom position
								GV_Axes.stAxisZ.lrAutoPosAbs:=GV_Tool_Magazine.stManipulator.lrZTunnelBottom;
							ENUM_Tunnel_Mode.BottomToTop: // Z top position
								GV_Axes.stAxisZ.lrAutoPosAbs:=GV_Tool_Magazine.stManipulator.lrZTunnelTop;
						END_CASE
						IF (GV_Axes.stAxisZ.lrAutoPosAbs=GV_Tool_Magazine.stManipulator.lrZTunnelBottom) OR (GV_Axes.stAxisZ.lrAutoPosAbs=GV_Tool_Magazine.stManipulator.lrZTunnelTop) THEN
							GV_Axes.stAxisZ.bAutoCmdAbs:=TRUE;
						ELSE
							GV_Axes.stAxisZ.bAutoCmdAbs:=FALSE;
						END_IF
						(*Log*)
							PRG_Log_WM.fbLogWM.M_Write_Log('FB_Manipulator_Tunnel : 3_Process : 2 : Start Z move');
						iSubStep:=3; // Next Step
		
					3: (* Wait Z move done *)
					   IF GV_Axes.stAxisZ.bAutoDone AND (NOT bZError) THEN
							GV_Axes.stAxisZ.bAutoCmdAbs:=FALSE;
							tonTimeout.IN:=FALSE;
							(*Log*)
								PRG_Log_WM.fbLogWM.M_Write_Log('FB_Manipulator_Tunnel : 2_Process : 3 : Z move done');
							bTunnelTravelDone:=TRUE;
							iSubStep:=0; // End SubStep
						ELSIF bZError THEN
							bError:=TRUE;
							udiErrorID:=33; // 33 = Step 3 SubStep 3 Error Axis Z
							GV_Axes.stAxisZ.bAutoCmdAbs:=FALSE;
							tonTimeout.IN:=FALSE;
							(*Log*)
								PRG_Log_WM.fbLogWM.M_Write_Log('FB_Manipulator_Tunnel : 3_Process=Error');
								PRG_Log_WM.fbLogWM.M_Write_Log(CONCAT('FB_Manipulator_Tunnel : ErrorID=',UDINT_TO_STRING(udiErrorID)));
							iSubStep:=0; // Stop SubStep
							iStep:=0; // Idle Step
						END_IF

					END_CASE
			
			IF bTunnelTravelDone THEN
				tonTimeout.IN:=FALSE;
				(*Log*)
					PRG_Log_WM.fbLogWM.M_Write_Log('FB_Manipulator_Tunnel : 2_Process : Done with success');
					PRG_Log_WM.fbLogWM.M_Write_Log('FB_Manipulator_Tunnel : 2_Process->0_Idle');
				iSubStep:=0; // End SubStep
				iStep:=0; // Idle Step
				bDone:=TRUE;
				bBusy:=FALSE;
			END_IF
			
			IF tonTimeout.Q AND tonTimeout.PT<>T#0S THEN
				bError:=TRUE;
				udiErrorID:=39; // 39 = Step 3 Error Timeout 9
				GV_Axes.stAxisZ.bAutoCmdAbs:=FALSE;
				GV_Axes.stAxisX.bAutoCmdAbs:=FALSE;
				GV_Axes.stAxisY.bAutoCmdAbs:=FALSE;
				tonTimeout.IN:=FALSE;
				(*Log*)
					PRG_Log_WM.fbLogWM.M_Write_Log('FB_Manipulator_Tunnel : 3_Process : Error');
					PRG_Log_WM.fbLogWM.M_Write_Log(CONCAT('FB_Manipulator_Tunnel : ErrorID = ',UDINT_TO_STRING(udiErrorID)));
				iSubStep:=0; // Stop SubStep
				iStep:=0; // Idle Step
			END_IF
			
	END_CASE

END_FUNCTION_BLOCK

// ---- 14_Log/03_POUs/01_PRGs/PRG_Log_WM.TcPOU
PROGRAM PRG_Log_WM
VAR
	(** FLAG **)
		bTest1 : BOOL ;
		bTest : BOOL ;
			
	(** FB **)
	 	fbLogWM : FB_LOG ;
END_VAR

//-----------------------------------------------------------------------------------------
//
//                  				PRG_Log_WM
//
//								Gestion des Log WM     			
//-----------------------------------------------------------------------------------------
//
//Auteur: G.GOETZ (inspired by S.MANTZER)
//Création: 04.02.2026
//Dernière modification : 04.02.2026 (G.GOETZ)
//       			
//-----------------------------------------------------------------------------------------
//
//     							Liste des modifications  	
//
// 04.02.2026 (G.GOETZ) -> Création		
//-----------------------------------------------------------------------------------------

(** FB **)
	fbLogWM(File_name:='WM_Log',File_number:=GV_Log.stLogWM.iFileNumber,Path_name:='C:\WM\Log\',File_management:=ENUM_Log_file_management.Automatic,Execute:=bTest,stLogData:=GV_Log.stLogWM);

(** WRITE TEXT IN LOG **)

	(* TEST *)
		(*Test 1*)
			GV_Log.aLogTrig[1](CLK:=bTest1);
			IF GV_Log.aLogTrig[1].Q THEN
				fbLogWM.M_Write_Log(strText:='TEST 1 : àè*156!ä£"+¨></*-_');
			END_IF

END_PROGRAM

// ---- 14_Log/03_POUs/02_FBs/FB_Log.TcPOU
FUNCTION_BLOCK FB_Log
VAR_INPUT
	File_name : STRING ; // File name without .CSV
	Path_name : STRING; // Path for file
	File_management : INT ; // File management :
										// 1:Automatic
										// 2:manual (with external start) 
										// 3:manual (with external start and file delete on start)
END_VAR
VAR_IN_OUT
	Execute : BOOL ; // Execute writing (not use in automatic mode)
	File_number : INT ; // File number
	stLogData : ST_LOG_DATA;
END_VAR
VAR
	FB_Write_log : FB_Write_DataToFile;
	Log_file_name : STRING ; // File name
	Temp_data : ARRAY[1..40000] OF BYTE;
	Init_data : ARRAY[1..40000] OF BYTE;
	Fill: UDINT ;
	Index : DINT;
	LENGTH : UDINT;
	LENGTH_FILE : UDINT;	
	SIZE : UDINT;
	SEPARATOR : STRING [10];
	END_OF_LINE : STRING [10];
	STEP : INT ;
	Save_timer : TON; // Timer for auto save
	File_delete : BOOL;
	Last_Log_date_time_new_file: INT;
END_VAR

//-----------------------------------------------------------------------------------------
//
//                  				FB_Log
//
//							Fonction pour les Log    			
//-----------------------------------------------------------------------------------------
//
//Auteur: G.GOETZ (inspired by S.MANTZER)
//Création: 04.02.2026
//Dernière modification : 04.02.2026 (G.GOETZ)
//       			
//-----------------------------------------------------------------------------------------
//
//     							Liste des modifications  	
//
// 04.02.2026 (G.GOETZ) -> Création		
//-----------------------------------------------------------------------------------------

Save_timer(IN:=NOT Save_timer.Q,PT:=T#60S);

// Buffer full
IF stLogData.iLineIndex>GV_Log.iMaxLog THEN
	stLogData.bBufferFull:=TRUE;
ELSE
	stLogData.bBufferFull:=FALSE;
END_IF

// Launch writing into file
IF STEP=0 THEN

	// Check file management mode
	CASE  File_management OF
		ENUM_Log_file_management.Automatic: // Automatic
			// Check if timer reach or check if buffer full
			IF (Save_timer.Q OR stLogData.bBufferFull) THEN 
				//check if new log file (each 24H)
				IF (GV_General.dtCurrentDateTime>(stLogData.dtLastLogDateTimeNewFile + T#24H)) THEN
					File_number:=File_number+1;
					File_delete:=TRUE;
					stLogData.dtLastLogDateTimeNewFile:=GV_General.dtCurrentDateTime;
					IF File_number>GV_Log.iMaxLogFile THEN
						File_number:=1;
					END_IF
				END_IF
				STEP:=1;
			END_IF	

		ENUM_Log_file_management.Manual: // Manual
			IF (Execute OR stLogData.bBufferFull) THEN
				STEP:=1;
				Execute:=FALSE;
			END_IF
			
		ENUM_Log_file_management.ManualWithDelete: // Manual with file delete
			IF Execute THEN
				STEP:=1;
				Execute:=FALSE;
				File_delete:=TRUE;
			END_IF					
	END_CASE
END_IF

// Preparing data and parameters
IF STEP=1 THEN
	Log_file_name :=Path_name;
	Log_file_name := CONCAT(Log_file_name,File_name);
	IF File_management=ENUM_Log_file_management.Automatic THEN
		Log_file_name := CONCAT(Log_file_name,INT_TO_STRING(File_number));
	END_IF
	Log_file_name := CONCAT(Log_file_name,'.CSV');
	Temp_data:=Init_data;
	Fill:=1;
	SEPARATOR:=';';
	END_OF_LINE:='$N';
	
		// Copy each log line in Array of bytes
		// Copy date and time
	FOR Index:=1 TO GV_Log.iMaxLog DO
		LENGTH:=INT_TO_UDINT(LEN(stLogData.aBufferLog[Index].strLogDateTime));
		IF LENGTH>0 THEN
			MEMCPY(destAddr:=ADR(Temp_data[Fill]),srcAddr:=ADR(stLogData.aBufferLog[Index].strLogDateTime),n:=LENGTH);
			Fill:=Fill+LENGTH;
			
			// Copy separator
			LENGTH:=INT_TO_UDINT(LEN(SEPARATOR));
			MEMCPY(destAddr:=ADR(Temp_data[Fill]),srcAddr:=ADR(SEPARATOR),n:=LENGTH);
			Fill:=Fill+LENGTH;
					
			// Copy log texte
			LENGTH:=INT_TO_UDINT(LEN(stLogData.aBufferLog[Index].strLogTxt));
			MEMCPY(destAddr:=ADR(Temp_data[Fill]),srcAddr:=ADR(stLogData.aBufferLog[Index].strLogTxt),n:=LENGTH);	
			Fill:=Fill+LENGTH;
					
			// Copy separator
			LENGTH:=INT_TO_UDINT(LEN(SEPARATOR));
			MEMCPY(destAddr:=ADR(Temp_data[Fill]),srcAddr:=ADR(SEPARATOR),n:=LENGTH);
			Fill:=Fill+LENGTH;
					
			// Copy End of line
			LENGTH:=INT_TO_UDINT(LEN(END_OF_LINE));
			MEMCPY(destAddr:=ADR(Temp_data[Fill]),srcAddr:=ADR(END_OF_LINE),n:=LENGTH);
			Fill:=Fill+LENGTH;
		END_IF		
	END_FOR
	// Reset WM log
	SIZE:=SIZEOF(stLogData.aBufferLog);
	LENGTH_FILE:=Fill-1;	
	MEMSET(destAddr:=ADR(stLogData.aBufferLog),fillByte:=0,n:=SIZE);
	stLogData.iLineIndex:=1;
	STEP:=2;
END_IF


// Write finished
IF FB_Write_log.bBusy THEN
	STEP:=0;
END_IF


FB_Write_log(sFilePath:=Log_file_name,DataToWrite:=ADR(Temp_data),DataToWriteLen:=LENGTH_FILE,bExecute:=STEP=2,With_file_delete:=File_delete);

METHOD M_Write_Log : BOOL
VAR_INPUT
	(** STRING **)
	strText : STRING(255 ); // Text to write in log
END_VAR
//-----------------------------------------------------------------------------------------
//
//                  				M_Write_Log
//
//						Méthode pour écritue dans le Log Buffer   			
//-----------------------------------------------------------------------------------------
//
//Auteur: G.GOETZ (inspired by S.MANTZER)
//Création: 04.02.2026
//Dernière modification : 04.02.2026 (G.GOETZ)
//       			
//-----------------------------------------------------------------------------------------
//
//     							Liste des modifications  	
//
// 04.02.2026 (G.GOETZ) -> Création		
//-----------------------------------------------------------------------------------------

(** WRITE DATA IN LOG BUFFER **)

	(* The warning can be disabled here as the user is aware of the risk that the reference may not be valid by checking its validity *)
		{warning disable C0371}
		
			IF PRG_MAIN.fbTime.systemTime.wYear<>1970 THEN
				IF stLogData.iLineIndex<=0 THEN
					stLogData.iLineIndex:=1;
				END_IF
				IF stLogData.iLineIndex<=GV_Log.iMaxLog THEN
					stLogData.aBufferLog[stLogData.iLineIndex].strLogDateTime:=sTime();
					stLogData.aBufferLog[stLogData.iLineIndex].strLogTxt:=strText;
					stLogData.iLineIndex:=stLogData.iLineIndex+1;
				END_IF
			END_IF
	
		{warning restore C0371}
	(* The warning may be restored at the end of the access area *)
END_METHOD

END_FUNCTION_BLOCK

// ---- 14_Log/03_POUs/02_FBs/FB_Write_DataToFile.TcPOU
FUNCTION_BLOCK FB_Write_DataToFile
VAR_INPUT
	sFilePath: STRING;
	DataToWrite: PVOID;
	DataToWriteLen: UDINT;	
	/// rising edge starts fb execution 
	bExecute: BOOL;
END_VAR
VAR_IN_OUT
	With_file_delete : BOOL; // File delete before writing
END_VAR
VAR_OUTPUT
	bBusy: BOOL;
	bError: BOOL;
	nErrId: UDINT;
END_VAR
VAR
	fbFileOpen: FB_FileOpen;
	fbFileDelete: FB_FileDelete;
	sNetID: STRING := '';
	sPathName: STRING := '';
	fbFileWrite: FB_FileWrite;
	fbFileClose: FB_FileClose;
	/// file handle of the destination file 
	hDestFile: UINT := 0;
	iSequence: INT := 0;
	RisingEdge: R_TRIG;
END_VAR

//-----------------------------------------------------------------------------------------
//
//                  			FB_Write_DataToFile
//
//							Fonction pour écrire les Log    			
//-----------------------------------------------------------------------------------------
//
//Auteur: G.GOETZ (inspired by S.MANTZER)
//Création: 04.02.2026
//Dernière modification : 04.02.2026 (G.GOETZ)
//       			
//-----------------------------------------------------------------------------------------
//
//     							Liste des modifications  	
//
// 04.02.2026 (G.GOETZ) -> Création		
//-----------------------------------------------------------------------------------------

RisingEdge(CLK:=bExecute);
IF RisingEdge.Q THEN
        IF NOT bBusy THEN
                bBusy := TRUE;
                bError:= FALSE;
                nErrId:=0;
                iSequence := 10;
                sPathName:='';
                hDestFile:=0;
        END_IF
END_IF

CASE iSequence OF
0:
	; (* do nothing *)

10:		// Reset Open block
		sPathName := sFilePath;
		fbFileOpen(	sNetId		:= sNetID,
				sPathName	:= sPathName,
				nMode		:=  FOPEN_MODEAPPEND OR FOPEN_MODEBINARY,
				ePath		:= PATH_GENERIC,
				bExecute	:= FALSE,
				tTimeout		:= T#5S);
		fbFileDelete(sNetId		:= sNetID,
				sPathName	:= sPathName,
				ePath		:= PATH_GENERIC,
				bExecute	:= FALSE,
				tTimeout		:= T#5S);
		iSequence := iSequence + 10;
		
20: // Open file or create if do not exit
		fbFileOpen(	sNetId		:= sNetID,
					sPathName	:= sPathName,
					nMode		:=  FOPEN_MODEAPPEND OR FOPEN_MODEBINARY,
					ePath		:= PATH_GENERIC,
					bExecute	:= TRUE,
					tTimeout		:= T#5S);
		iSequence := iSequence + 10;

30: (* loop in this state until not bBusy *)
	 fbFileOpen();
	IF (NOT fbFileOpen.bBusy) AND (NOT fbFileOpen.bError) THEN
		hDestFile	:= fbFileOpen.hFile;
		fbFileOpen(	sNetId		:= sNetID,
					sPathName	:= sPathName,
					nMode		:= FOPEN_MODEAPPEND OR FOPEN_MODEBINARY,
					ePath		:= PATH_GENERIC,
					bExecute	:= FALSE,
					tTimeout		:= T#5S);
			iSequence := 60;
		// Check if file delete need
		// Closing file before delete
		IF With_file_delete THEN
			fbFileClose(	sNetId		:= sNetID,
				hFile		:= hDestFile,
				bExecute	:= TRUE,
				tTimeout		:=  T#5S);
			iSequence := 40;
		END_IF
	ELSE	(* handle error *)
		IF fbFileOpen.bError THEN
		 	iSequence :=900;
		END_IF
	END_IF

40:	// Delete file before writing
	 fbFileClose();
	IF (NOT fbFileClose.bBusy) AND (NOT fbFileClose.bError) THEN
		fbFileClose(	sNetId		:= sNetID,
				hFile		:= hDestFile,
				bExecute	:= FALSE,
				tTimeout		:=  T#5S);
		fbFileDelete(sNetId		:= sNetID,
					sPathName	:= sPathName,
					ePath		:= PATH_GENERIC,
					bExecute	:= TRUE,
					tTimeout		:= T#5S);
		iSequence := iSequence + 10;
	ELSE	(* handle error *)
		IF fbFileClose.bError THEN
		 	iSequence :=900;
		END_IF
	END_IF

50:	// File deleted, create new
	 fbFileDelete();
	IF (NOT fbFileDelete.bBusy) AND (NOT fbFileDelete.bError) THEN
		fbFileDelete(sNetId		:= sNetID,
				sPathName	:= sPathName,
				ePath		:= PATH_GENERIC,
				bExecute	:= FALSE,
				tTimeout		:= T#5s);
		// File deleted
		With_file_delete:=FALSE;
		iSequence := 10;
	ELSE	(* handle error *)
		IF fbFileDelete.bError THEN
		 	iSequence :=900;
		END_IF
	END_IF
	
60:	fbFileWrite(	sNetId		:= sNetID,
				hFile		:= hDestFile,
				pWriteBuff	:= DataToWrite,
				cbWriteLen	:= DataToWriteLen,
				bExecute	:= FALSE,
				tTimeout		:= T#5S  );
	iSequence :=90;

90:
	fbFileWrite(	sNetId		:= sNetID,
				hFile		:= hDestFile,
				pWriteBuff	:= DataToWrite,
				cbWriteLen	:= DataToWriteLen,
				bExecute	:= TRUE,
				tTimeout		:= T#5S  );
	iSequence := iSequence + 10;


100: (* loop in this state until not bBusy *)
	fbFileWrite();
	IF (NOT fbFileWrite.bBusy) AND (NOT fbFileWrite.bError) THEN
		fbFileWrite(	sNetId		:= sNetID,
					hFile		:= hDestFile,
					pWriteBuff	:= DataToWrite,
					cbWriteLen	:= DataToWriteLen,
					bExecute	:= FALSE,
					tTimeout		:= T#5S  );
		iSequence := 110;
	ELSE	(* handle error *)
		IF fbFileWrite.bError THEN
		 	iSequence :=900;
		END_IF
	END_IF

110:	fbFileClose(	sNetId		:= sNetID,
				hFile		:= hDestFile,
				bExecute	:= FALSE,
				tTimeout		:=  T#5S);
	iSequence :=120;

120:
	fbFileClose(	sNetId		:= sNetID,
				hFile		:= hDestFile,
				bExecute	:= TRUE,
				tTimeout		:=  T#5S);
	iSequence := iSequence + 10;

130: (* loop in this state until not bBusy *)
	fbFileClose();
	IF (NOT fbFileClose.bBusy) AND (NOT fbFileClose.bError) THEN
		fbFileClose(	sNetId		:= sNetID,
					hFile		:= hDestFile,
					bExecute	:= FALSE,
					tTimeout		:=  T#5S);
		iSequence := 140;
	ELSE	(* handle error *)
		IF fbFileClose.bError THEN
		 	iSequence :=900;
		END_IF
	END_IF

140:
		bBusy:=FALSE;
		iSequence := 0;


900:
	(* additional code to log the error, either  fbFileOpen.bError,fbFileWrite.bError or  fbFileClose.bError *)
	(* close the file if it is open *)
	IF hDestFile<>0 THEN
		fbFileClose(	sNetId		:= sNetID,
					hFile		:= hDestFile,
					bExecute	:= TRUE,
					tTimeout		:=  T#5S);
			iSequence := iSequence + 10;
	ELSE
		iSequence := 999;
	END_IF

910: (* loop in this state until not bBusy *)
	IF (NOT fbFileClose.bBusy) AND (NOT fbFileClose.bError) THEN
		fbFileClose(	sNetId		:= sNetID,
					hFile		:= hDestFile,
					bExecute	:= FALSE,
					tTimeout		:=  T#5s);
		iSequence := 999;
	ELSE	(* handle error *)
		IF fbFileClose.bError THEN
		 	iSequence :=999;
		END_IF
	END_IF

999:

		bBusy:=FALSE;
		iSequence := 0;


END_CASE

END_FUNCTION_BLOCK

// ---- 14_Log/03_POUs/02_FBs/sTime.TcPOU
FUNCTION sTime : STRING
VAR_INPUT
END_VAR
VAR
	(** STRING **)
		strDateTime : STRING;
END_VAR

//-----------------------------------------------------------------------------------------
//
//                  				sTime
//
//							Transformation Date et Heure    			
//-----------------------------------------------------------------------------------------
//
//Auteur: G.GOETZ (inspired by S.MANTZER)
//Création: 04.02.2026
//Dernière modification : 04.02.2026 (G.GOETZ)
//       			
//-----------------------------------------------------------------------------------------
//
//     							Liste des modifications  	
//
// 04.02.2026 (G.GOETZ) -> Création		
//-----------------------------------------------------------------------------------------

(** Return actual date and time in string format, with ; separator between date and hour* *)
	strDateTime := SYSTEMTIME_TO_STRING(PRG_MAIN.fbTime.systemTime);
	
	sTime := CONCAT( LEFT(STR:=strDateTime, SIZE := 10 ) ,  CONCAT( ';', DELETE( STR:= strDateTime, LEN:= 11, POS:= 1) )  );
	sTime := REPLACE(STR1:=sTime,STR2:= ';',L:= 1,P:= 20);

END_FUNCTION

// ---- 08_Cycle/03_POUs/02_FBs/FB_01_Action_PickToolMagazine.TcPOU
FUNCTION_BLOCK FB_01_Action_PickToolMagazine
VAR_INPUT
	(** SETUP ST **)
		stToolLocation : ST_Tool_Location ; // Tool_Location structure of the Tool to Pick
		
	(** SETUP TIME **)
		(*Manipulator Gripper mvmnt*)
			tMouvementGripperOpen : TIME ; // Value of the manipulator gripper open mouvement duration (fbGripper)
			tMouvementGripperClose : TIME ; // Value of the manipulator gripper close mouvement duration (fbGripper)
		(*Tunnel*)
			tTunnelTimeout : TIME ; // Value of the timeout for travel the tunnel
		(*Step 2*)
			tMove2Timeout : TIME ; // Value of the timeout for Step 2
		(*Step 4*)
			tMove4Timeout : TIME ; // Value of the timeout for Step 4
		(*Step 6*)
			tMove6Timeout : TIME ; // Value of the timeout for Step 6
		(*Step 8*)
			tMove8Timeout : TIME ; // Value of the timeout for Step 8

	(** SETUP LREAL **)
		lrZToolOffset : LREAL ; // Z Offset above the tool

	(** SETUP FLAG **)
		bCheckSensorManipulatorGripper : BOOL ; // Check the manipulator gripper sensor at the beginning
		(*Gripper*)
			bCheckSensorGripperOpen : BOOL ; // Check the manipulator gripper sensor after open (fbGripper)
			bCheckSensorGripperClose : BOOL ; // Check the manipulator gripper sensor after close (fbGripper)
			
	(** PROCESS FLAG **)
		bInit : BOOL ;  // Init the Fb
	    bStart : BOOL ; // Start the Fb
END_VAR
VAR_OUTPUT
	(** PROCESS UUDINT **)
		udiErrorID : UDINT ; // Fb Error ID
		
	(** PROCESS FLAG **)
		bBusy  : BOOL ; // Fb is Busy
		bDone  : BOOL ; // Fb is Done
		bError : BOOL ; // Fb in Error
END_VAR
VAR_IN_OUT
END_VAR	
VAR
	(** SETUP ENUM **)
		(*Gripper*)
			eGripperMode : ENUM_Gripper_Mode; // Gripper mode for gripper mouvement (fbGripper)
		(*Tunnel*)
			eTunnelMode : ENUM_Tunnel_Mode; // Tunnel mode for travel (fbTunnel)

	(** SETUP TIME **)
		(*Gripper*)
			tGripperTime : TIME ; // Mouvement duration for gripper mouvement (fbGripper)
	
	(** SETUP FLAG **)
		(*Gripper*)
			bGripperSensor : BOOL ; // Sensor check for gripper mouvement (fbGripper)
		
	(** PROCESS STRING **)
		strTextLog : STRING ; // Text to Log
		
	(** PROCESS LREAL **)
		
	(** PROCESS INT **)
		iStep  : INT := 0 ; // Step of the Fb
		iSubStep : INT := 0 ; // SubStep of the Fb
		iPrevStep : INT := 0 ; // Previous Step of the Fb
		iPrevSubStep : INT := 0 ; // Previous Subtep of the Fb
		
	(** PROCESS FLAG + R_TRIG **)
		rtInit : R_TRIG ; // FB Init at rising edge
		rtStart : R_TRIG ; // FB Start at rising edge
		(*Tunnel*)
			bTunnelTravel : BOOL ; // Need to travel the tunnel
		bXError : BOOL ; // Axis X Error
		bYError : BOOL ; // Axis Y Error
		bZError : BOOL ; // Axis Z Error
		bArmError : BOOL ; // Axis Arm Error
		
	(** FB **)
		(*Gripper*)
			fbGripper : FB_Manipulator_Gripper ;
		(*Tunnel*)
			fbTunnel : FB_Manipulator_Tunnel ;
		(*Step 2*)
			tonTimeoutMove2 : TON ; // TON timeout for the Step 2
		(*Step 4*)
			tonTimeoutMove4 : TON ; // TON timeout for the Step 4
		(*Step 6*)
			tonTimeoutMove6 : TON ; // TON timeout for the Step 6
		(*Step 8*)
			tonTimeoutMove8 : TON ; // TON timeout for the Step 8
END_VAR

//-----------------------------------------------------------------------------------------
//
//                  			FB_01_Action_PickToolMagazine
//
//						Management of the pick tool on the magazine
//-----------------------------------------------------------------------------------------
//
//Auteur: G.GOETZ
//Création: 04.02.2026
//Dernière modification : 08.04.2026 (G.GOETZ)
//       			
//-----------------------------------------------------------------------------------------
//
//     							Liste des modifications  	
//
// 04.02.2026 (G.GOETZ) -> Création
// 08.04.2026 (G.GOETZ) -> Ajout Init + Modification du cycle
//-----------------------------------------------------------------------------------------

(** FB CALL **)
	rtInit(CLK:=bInit);
	rtStart(CLK:=bStart);
	
	tonTimeoutMove2();
	tonTimeoutMove4();
	tonTimeoutMove6();
	tonTimeoutMove8();
	fbGripper( // Call Gripper mouvement
			eGripperMode:=eGripperMode,
			tMouvementDuration:=tGripperTime,
			bSensorCheck:=bGripperSensor
			);
	fbTunnel( // Call Tunnel travel
			eTunnelMode:=eTunnelMode,
			tTimeout:=tTunnelTimeout
			);

(** AXIS ERRORS **)
	bXError:=(GV_Axes.stAxisX.stDriveAx8206.AxisRef.Status.Error OR GV_Axes.stAxisX.stDriveAx8206.AxisRef.Status.ErrorStop OR GV_Axes.stAxisX.stDriveAx8206.AxisRef.Status.ErrorID<>0);
	bYError:=(GV_Axes.stAxisY.stDriveAx8206.AxisRef.Status.Error OR GV_Axes.stAxisY.stDriveAx8206.AxisRef.Status.ErrorStop OR GV_Axes.stAxisY.stDriveAx8206.AxisRef.Status.ErrorID<>0);
	bZError:=(GV_Axes.stAxisZ.stDriveAx8206.AxisRef.Status.Error OR GV_Axes.stAxisZ.stDriveAx8206.AxisRef.Status.ErrorStop OR GV_Axes.stAxisZ.stDriveAx8206.AxisRef.Status.ErrorID<>0);
	bArmError:=(GV_Axes.stAxisArm.stDriveAx8206.AxisRef.Status.Error OR GV_Axes.stAxisArm.stDriveAx8206.AxisRef.Status.ErrorStop OR GV_Axes.stAxisArm.stDriveAx8206.AxisRef.Status.ErrorID<>0);

(** INIT **)
	IF (rtinit.Q OR bInit) AND (NOT bStart) THEN
		iStep:=0;
		bInit:=FALSE;
	END_IF
	
(** STEPS **)
    CASE iStep OF
		
        0: (* Step 0 = Idle + Check *)
            bBusy:=FALSE;
            bDone:=FALSE;
			bError:=FALSE;
			udiErrorID:=0;
			iSubStep:=0;
			
			tonTimeoutMove2.IN:=FALSE;
			tonTimeoutMove4.IN:=FALSE;
			tonTimeoutMove6.IN:=FALSE;
			tonTimeoutMove8.IN:=FALSE;
			
			GV_Axes.stAxisX.bAutoCmdAbs:=FALSE;
			GV_Axes.stAxisY.bAutoCmdAbs:=FALSE;
			GV_Axes.stAxisZ.bAutoCmdAbs:=FALSE;
			
			fbGripper.bInit:=TRUE;
			fbTunnel.bInit:=TRUE;
			
			bTunnelTravel:=FALSE;
			
			(* Idle->Start *)
				IF rtStart.Q AND (NOT bInit) THEN
					bBusy:=TRUE;
					(*Log*)
						(*Location*)
							strTextLog:=INT_TO_STRING(stToolLocation.iAbsLocationNumber);
							PRG_Log_WM.fbLogWM.M_Write_Log(CONCAT('FB_01_Action_PickToolMagazine : 0_Idle : Tool Location Abs = ',strTextLog));
							strTextLog:=INT_TO_STRING(stToolLocation.iRelLocationNumber);
							PRG_Log_WM.fbLogWM.M_Write_Log(CONCAT('FB_01_Action_PickToolMagazine : 0_Idle : Tool Location Rel = ',strTextLog));
							strTextLog:=DINT_TO_STRING(stToolLocation.stToolParam.Number);
							PRG_Log_WM.fbLogWM.M_Write_Log(CONCAT('FB_01_Action_PickToolMagazine : 0_Idle : Tool Number = ',strTextLog));
						(*Sensor Check Manipulator*)
							IF bCheckSensorManipulatorGripper THEN
								strTextLog:='With';
							ELSE
								strTextLog:='Without';
							END_IF
							PRG_Log_WM.fbLogWM.M_Write_Log(CONCAT('FB_01_Action_PickToolMagazine : 0_Idle : Sensor Manipulator memory Check = ',strTextLog));
						(*Z Tool Offset*)
							strTextLog:=LREAL_TO_STRING(lrZToolOffset);
							PRG_Log_WM.fbLogWM.M_Write_Log(CONCAT('FB_01_Action_PickToolMagazine : 0_Idle : Z Tool Offset = ',strTextLog));
						(*Timeout Step 2_AboveLocation*)
							strTextLog:=TIME_TO_STRING(tMove2Timeout);
							PRG_Log_WM.fbLogWM.M_Write_Log(CONCAT('FB_01_Action_PickToolMagazine : 0_Idle : Timeout Step : 2_AboveLocation = ',strTextLog));
						(*Timeout Step 4_Location*)
							strTextLog:=TIME_TO_STRING(tMove4Timeout);
							PRG_Log_WM.fbLogWM.M_Write_Log(CONCAT('FB_01_Action_PickToolMagazine : 0_Idle : Timeout Step : 4_Location = ',strTextLog));
						(*Timeout Step 6_FrontLocation*)
							strTextLog:=TIME_TO_STRING(tMove6Timeout);
							PRG_Log_WM.fbLogWM.M_Write_Log(CONCAT('FB_01_Action_PickToolMagazine : 0_Idle : Timeout Step : 6_FrontLocation = ',strTextLog));
						(*Timeout Step 8_PositionTransferArm*)
							strTextLog:=TIME_TO_STRING(tMove8Timeout);
							PRG_Log_WM.fbLogWM.M_Write_Log(CONCAT('FB_01_Action_PickToolMagazine : 0_Idle : Timeout Step : 8_PositionTransferArm = ',strTextLog));

					(*Check Manipulator*)
					IF (NOT GV_CNC.stFanucData.stMagazineCNC.boOpenManipulatorGripper) THEN // Gripper Close
						(*Log*)
							PRG_Log_WM.fbLogWM.M_Write_Log('FB_01_Action_PickToolMagazine : 0_Idle : Manipulator Gripper Check = OK');
							PRG_Log_WM.fbLogWM.M_Write_Log('FB_01_Action_PickToolMagazine : 0_Idle : Manipulator Gripper = CLOSE');
						IF (NOT GV_Tool_Magazine.stManipulator.bToolPresenceMemory) THEN // Gripper Memory
							(*Log*)
								PRG_Log_WM.fbLogWM.M_Write_Log('FB_01_Action_PickToolMagazine : 0_Idle : Manipulator memory Check = OK');
							IF bCheckSensorManipulatorGripper THEN
								IF (NOT GV_IO.diToolPresenceCone) THEN // Gripper Sensor
									(*Log*)
										PRG_Log_WM.fbLogWM.M_Write_Log('FB_01_Action_PickToolMagazine : 0_Idle : Manipulator sensor Check = FALSE = OK');
								ELSE
									bError:=TRUE;
									udiErrorID:=003; // 003 = Step 0 Error Manipulator Sensor Check 03
									(*Log*)
										PRG_Log_WM.fbLogWM.M_Write_Log('FB_01_Action_PickToolMagazine : 0_Idle : Manipulator sensor Check = TRUE = NOK');
										PRG_Log_WM.fbLogWM.M_Write_Log('FB_01_Action_PickToolMagazine : 0_Idle=Error');
										PRG_Log_WM.fbLogWM.M_Write_Log(CONCAT('FB_01_Action_PickToolMagazine : ErrorID=',UDINT_TO_STRING(udiErrorID)));
									iStep:=0; // Idle Step
								END_IF
							ELSE
								(*Log*)
									PRG_Log_WM.fbLogWM.M_Write_Log('FB_01_Action_PickToolMagazine : 0_Idle : Manipulator sensor Check : Not controlled');
							END_IF
						ELSE
							bError:=TRUE;
							udiErrorID:=002; // 002 = Step 0 Error Manipulator Memory Check 02
							(*Log*)
								PRG_Log_WM.fbLogWM.M_Write_Log('FB_01_Action_PickToolMagazine : 0_Idle : Manipulator memory Check = NOK');
								PRG_Log_WM.fbLogWM.M_Write_Log('FB_01_Action_PickToolMagazine : 0_Idle : Manipulator memory = Presence');
								strTextLog:=INT_TO_STRING(GV_Tool_Magazine.stManipulator.iAbsLocationNumberMemory);
								PRG_Log_WM.fbLogWM.M_Write_Log(CONCAT('FB_01_Action_PickToolMagazine : 0_Idle : Manipulator memory Location Number Abs = ',strTextLog));
								strTextLog:=INT_TO_STRING(GV_Tool_Magazine.stManipulator.iRelLocationNumberMemory);
								PRG_Log_WM.fbLogWM.M_Write_Log(CONCAT('FB_01_Action_PickToolMagazine : 0_Idle : Manipulator memory Location Number Rel = ',strTextLog));
								PRG_Log_WM.fbLogWM.M_Write_Log('FB_01_Action_PickToolMagazine : 0_Idle=Error');
								PRG_Log_WM.fbLogWM.M_Write_Log(CONCAT('FB_01_Action_PickToolMagazine : ErrorID=',UDINT_TO_STRING(udiErrorID)));
							iStep:=0; // Idle Step
						END_IF
					ELSE
						bError:=TRUE;
						udiErrorID:=001; // 001 = Step 0 Error Manipulator Gripper Open 01
						(*Log*)
							PRG_Log_WM.fbLogWM.M_Write_Log('FB_01_Action_PickToolMagazine : 0_Idle : Manipulator Gripper Check = NOK');
							PRG_Log_WM.fbLogWM.M_Write_Log('FB_01_Action_PickToolMagazine : 0_Idle : Manipulator Gripper = OPEN');
							PRG_Log_WM.fbLogWM.M_Write_Log('FB_01_Action_PickToolMagazine : 0_Idle=Error');
							PRG_Log_WM.fbLogWM.M_Write_Log(CONCAT('FB_01_Action_PickToolMagazine : ErrorID=',UDINT_TO_STRING(udiErrorID)));
						iStep:=0; // Idle Step
					END_IF
					
					IF (NOT bError) THEN
						(*Log*)
							PRG_Log_WM.fbLogWM.M_Write_Log('FB_01_Action_PickToolMagazine : 0_Idle->1_Tunnel');
						iStep:=1; // Next Step
					END_IF
					
				END_IF
				
		1: (* Step 1 = Tunnel passage (if needed) *)
			IF (NOT bTunnelTravel) THEN
				IF (stToolLocation.ePositionMag=ENUM_Position_Magazine.Bottom AND GV_Tool_Magazine.stManipulator.ePositionMag=ENUM_Position_Magazine.Bottom) OR (stToolLocation.ePositionMag=ENUM_Position_Magazine.Top AND GV_Tool_Magazine.stManipulator.ePositionMag=ENUM_Position_Magazine.Top) THEN
					bTunnelTravel:=FALSE;
					(*Log*)
						PRG_Log_WM.fbLogWM.M_Write_Log('FB_01_Action_PickToolMagazine : 1_Tunnel : No Need to Travel');
						PRG_Log_WM.fbLogWM.M_Write_Log('FB_01_Action_PickToolMagazine : 1_Tunnel->2_AboveLocation');
					iStep:=2; // Next Step
				END_IF	
				IF stToolLocation.ePositionMag=ENUM_Position_Magazine.Bottom AND GV_Tool_Magazine.stManipulator.ePositionMag=ENUM_Position_Magazine.Top THEN
					eTunnelMode:=ENUM_Tunnel_MODE.TopToBottom;
					bTunnelTravel:=TRUE;
					(*Log*)
						PRG_Log_WM.fbLogWM.M_Write_Log('FB_01_Action_PickToolMagazine : 1_Tunnel : Need to Travel Top->Bottom');
				END_IF
				IF stToolLocation.ePositionMag=ENUM_Position_Magazine.Top AND GV_Tool_Magazine.stManipulator.ePositionMag=ENUM_Position_Magazine.Bottom THEN
					eTunnelMode:=ENUM_Tunnel_MODE.BottomToTop;
					bTunnelTravel:=TRUE;
					(*Log*)
						PRG_Log_WM.fbLogWM.M_Write_Log('FB_01_Action_PickToolMagazine : 1_Tunnel : Need to Travel Bottom->Top');
				END_IF			
				IF stToolLocation.ePositionMag<>ENUM_Position_Magazine.Unknow AND GV_Tool_Magazine.stManipulator.ePositionMag=ENUM_Position_Magazine.Unknow THEN // Manipulator Unknow position
					bError:=TRUE;
					udiErrorID:=101; // 101 = Step 1 Error Tunnel 01
					bTunnelTravel:=FALSE;
					(*Log*)
						PRG_Log_WM.fbLogWM.M_Write_Log('FB_01_Action_PickToolMagazine : 1_Tunnel=Error');
						PRG_Log_WM.fbLogWM.M_Write_Log(CONCAT('FB_01_Action_PickToolMagazine : ErrorID=',UDINT_TO_STRING(udiErrorID)));
					iStep:=0; // Idle Step
				END_IF
				IF stToolLocation.ePositionMag=ENUM_Position_Magazine.Unknow AND GV_Tool_Magazine.stManipulator.ePositionMag<>ENUM_Position_Magazine.Unknow THEN // ToolLocation Unknow position
					bError:=TRUE;
					udiErrorID:=102; // 102 = Step 1 Error Tunnel 02
					bTunnelTravel:=FALSE;
					(*Log*)
						PRG_Log_WM.fbLogWM.M_Write_Log('FB_01_Action_PickToolMagazine : 1_Tunnel=Error');
						PRG_Log_WM.fbLogWM.M_Write_Log(CONCAT('FB_01_Action_PickToolMagazine : ErrorID=',UDINT_TO_STRING(udiErrorID)));
					iStep:=0; // Idle Step
				END_IF
				IF stToolLocation.ePositionMag=ENUM_Position_Magazine.Unknow AND GV_Tool_Magazine.stManipulator.ePositionMag=ENUM_Position_Magazine.Unknow THEN // ToolLocation AND Manipulator Unknow position
					bError:=TRUE;
					udiErrorID:=103; // 103 = Step 1 Error Tunnel 03
					bTunnelTravel:=FALSE;
					(*Log*)
						PRG_Log_WM.fbLogWM.M_Write_Log('FB_01_Action_PickToolMagazine : 1_Tunnel=Error');
						PRG_Log_WM.fbLogWM.M_Write_Log(CONCAT('FB_01_Action_PickToolMagazine : ErrorID=',UDINT_TO_STRING(udiErrorID)));
					iStep:=0; // Idle Step
				END_IF
			END_IF
			
			IF bTunnelTravel AND (NOT fbTunnel.bStart) AND (NOT fbTunnel.bInit) AND (NOT fbTunnel.bBusy) THEN // Tunnel Start
				fbTunnel.bStart:=TRUE;
			END_IF
			IF fbTunnel.bDone AND (NOT fbTunnel.bError) THEN // Tunnel Done
				fbTunnel.bStart:=FALSE;
				bTunnelTravel:=FALSE;
				(*Log*)
					PRG_Log_WM.fbLogWM.M_Write_Log('FB_01_Action_PickToolMagazine : 1_Tunnel->2_AboveLocation');
				iStep:=2; // Next Step
			ELSIF fbTunnel.bError THEN // Tunnel Error
				bError:=TRUE;
				udiErrorID:=100+fbTunnel.udiErrorID; // 1xx = Step 1 Error + Error xx fbTunnel
				fbTunnel.bStart:=FALSE;
				bTunnelTravel:=FALSE;
				(*Log*)
					PRG_Log_WM.fbLogWM.M_Write_Log('FB_01_Action_PickToolMagazine : 1_Tunnel=Error');
					PRG_Log_WM.fbLogWM.M_Write_Log(CONCAT('FB_01_Action_PickToolMagazine : ErrorID=',UDINT_TO_STRING(udiErrorID)));
				iStep:=0; // Idle Step
			END_IF
			
		2: (* Step 2 = Move the manipulator above the tool/location (YHome->(XFirst)->ZOffset->X->Y) *)
			tonTimeoutMove2.PT:=tMove2Timeout;
			tonTimeoutMove2.IN:=TRUE;
			
			CASE iSubStep OF

				0: (* Start YHome move *)
					GV_Axes.stAxisY.lrAutoPosAbs:=GV_Tool_Magazine.stManipulator.lrYHome;
					GV_Axes.stAxisY.bAutoCmdAbs:=TRUE;
					(*Log*)
						PRG_Log_WM.fbLogWM.M_Write_Log('FB_01_Action_PickToolMagazine : 2_AboveLocation : 0 : Start YHome move');
					iSubStep:=1; // Next SubStep

				1: (* Wait YHome move done *)
				   IF GV_Axes.stAxisY.bAutoDone AND (NOT bYError) THEN
						GV_Axes.stAxisY.bAutoCmdAbs:=FALSE;
						(*Log*)
							PRG_Log_WM.fbLogWM.M_Write_Log('FB_01_Action_PickToolMagazine : 2_AboveLocation : 1 : YHome move done');
							(*Top*)
								IF GV_Tool_Magazine.stManipulator.ePositionMag=ENUM_Position_Magazine.Top THEN
									IF GV_Tool_Magazine.stManipulator.lrXPosition<GV_Tool_Magazine.lrXFirstLocationTop THEN
										(*Log*)
											PRG_Log_WM.fbLogWM.M_Write_Log('FB_01_Action_PickToolMagazine : 2_AboveLocation : 1->2 : XFirstTop');
										//iSubStep:=2; // Next SubStep // ICI ; revoir, peut-être même ajouter ZLowestRackTop avant le XFirst car si part direct en XFirst depuis la position transfer ver bras alors tape dans le bras !
										iSubStep:=4; // Next SubStep
									ELSE
										(*Log*)
											PRG_Log_WM.fbLogWM.M_Write_Log('FB_01_Action_PickToolMagazine : 2_AboveLocation : 1->4 : ZOffset');
										iSubStep:=4; // Next SubStep
									END_IF
								END_IF
							(*Bottom*)
								IF GV_Tool_Magazine.stManipulator.ePositionMag=ENUM_Position_Magazine.Bottom THEN
									IF GV_Tool_Magazine.stManipulator.lrXPosition<GV_Tool_Magazine.lrXFirstLocationBottom THEN
										(*Log*)
											PRG_Log_WM.fbLogWM.M_Write_Log('FB_01_Action_PickToolMagazine : 2_AboveLocation : 1->2 : XFirstBottom');
										iSubStep:=2; // Next SubStep
									ELSE
										(*Log*)
											PRG_Log_WM.fbLogWM.M_Write_Log('FB_01_Action_PickToolMagazine : 2_AboveLocation : 1->4 : ZOffset');
										iSubStep:=4; // Next SubStep
									END_IF
								END_IF
					ELSIF bYError THEN
						bError:=TRUE;
						udiErrorID:=211; // 211 = Step 2 SubStep 1 Error Axis Y 1
						GV_Axes.stAxisY.bAutoCmdAbs:=FALSE;
						tonTimeoutMove2.IN:=FALSE;
						(*Log*)
							PRG_Log_WM.fbLogWM.M_Write_Log('FB_01_Action_PickToolMagazine : 2_AboveLocation=Error');
							PRG_Log_WM.fbLogWM.M_Write_Log(CONCAT('FB_01_Action_PickToolMagazine : ErrorID=',UDINT_TO_STRING(udiErrorID)));
						iSubStep:=0; // Stop SubStep
						iStep:=0; // Idle Step
					END_IF

				2: (* Start XFirst move *)
					IF GV_Tool_Magazine.stManipulator.ePositionMag=ENUM_Position_Magazine.Top THEN
						GV_Axes.stAxisX.lrAutoPosAbs:=GV_Tool_Magazine.lrXFirstLocationTop;
						(*Log*)
							PRG_Log_WM.fbLogWM.M_Write_Log('FB_01_Action_PickToolMagazine : 2_AboveLocation : 2 : Start XFisrtTop move');
					END_IF
					IF GV_Tool_Magazine.stManipulator.ePositionMag=ENUM_Position_Magazine.Bottom THEN
						GV_Axes.stAxisX.lrAutoPosAbs:=GV_Tool_Magazine.lrXFirstLocationBottom;
						(*Log*)
							PRG_Log_WM.fbLogWM.M_Write_Log('FB_01_Action_PickToolMagazine : 2_AboveLocation : 2 : Start XFisrtBottom move');
					END_IF
					GV_Axes.stAxisX.bAutoCmdAbs:=TRUE;
					iSubStep:=3; // Next SubStep

				3: (* Wait XFirst move done *)
				   IF GV_Axes.stAxisX.bAutoDone AND (NOT bXError) THEN
						GV_Axes.stAxisX.bAutoCmdAbs:=FALSE;
						(*Log*)
							PRG_Log_WM.fbLogWM.M_Write_Log('FB_01_Action_PickToolMagazine : 2_AboveLocation : 3 : XFirst move done');
						iSubStep:=4; // Next SubStep
					ELSIF bXError THEN
						bError:=TRUE;
						udiErrorID:=231; // 231 = Step 2 SubStep 3 Error Axis X 1
						GV_Axes.stAxisX.bAutoCmdAbs:=FALSE;
						tonTimeoutMove2.IN:=FALSE;
						(*Log*)
							PRG_Log_WM.fbLogWM.M_Write_Log('FB_01_Action_PickToolMagazine : 2_AboveLocation=Error');
							PRG_Log_WM.fbLogWM.M_Write_Log(CONCAT('FB_01_Action_PickToolMagazine : ErrorID=',UDINT_TO_STRING(udiErrorID)));
						iSubStep:=0; // Stop SubStep
						iStep:=0; // Idle Step
					END_IF

				4: (* Start ZOffset move *)
					GV_Axes.stAxisZ.lrAutoPosAbs:=stToolLocation.lrZcoord+lrZToolOffset;
					GV_Axes.stAxisZ.bAutoCmdAbs:=TRUE;
					(*Log*)
						PRG_Log_WM.fbLogWM.M_Write_Log('FB_01_Action_PickToolMagazine : 2_AboveLocation : 4 : Start ZOffset move');
					iSubStep:=5; // Next SubStep

				5: (* Wait ZOffset move done *)
				   IF GV_Axes.stAxisZ.bAutoDone AND (NOT bZError) THEN
						GV_Axes.stAxisZ.bAutoCmdAbs:=FALSE;
						(*Log*)
							PRG_Log_WM.fbLogWM.M_Write_Log('FB_01_Action_PickToolMagazine : 2_AboveLocation : 5 : ZOffset move done');
						iSubStep:=6; // Next SubStep
					ELSIF bZError THEN
						bError:=TRUE;
						udiErrorID:=251; // 251 = Step 2 SubStep 5 Error Axis Z 1
						GV_Axes.stAxisZ.bAutoCmdAbs:=FALSE;
						tonTimeoutMove2.IN:=FALSE;
						(*Log*)
							PRG_Log_WM.fbLogWM.M_Write_Log('FB_01_Action_PickToolMagazine : 2_AboveLocation=Error');
							PRG_Log_WM.fbLogWM.M_Write_Log(CONCAT('FB_01_Action_PickToolMagazine : ErrorID=',UDINT_TO_STRING(udiErrorID)));
						iSubStep:=0; // Stop SubStep
						iStep:=0; // Idle Step
					END_IF
					
				6: (* Start X move *)
					GV_Axes.stAxisX.lrAutoPosAbs:=stToolLocation.lrXcoord;
					GV_Axes.stAxisX.bAutoCmdAbs:=TRUE;
					(*Log*)
						PRG_Log_WM.fbLogWM.M_Write_Log('FB_01_Action_PickToolMagazine : 2_AboveLocation : 6 : Start X move');
					iSubStep:=7; // Next SubStep

				7: (* Wait X move done *)
				   IF GV_Axes.stAxisX.bAutoDone AND (NOT bXError) THEN
						GV_Axes.stAxisX.bAutoCmdAbs:=FALSE;
						(*Log*)
							PRG_Log_WM.fbLogWM.M_Write_Log('FB_01_Action_PickToolMagazine : 2_AboveLocation : 7 : X move done');
						iSubStep:=8; // Next SubStep
					ELSIF bXError THEN
						bError:=TRUE;
						udiErrorID:=271; // 271 = Step 2 SubStep 7 Error Axis X 1
						GV_Axes.stAxisX.bAutoCmdAbs:=FALSE;
						tonTimeoutMove2.IN:=FALSE;
						(*Log*)
							PRG_Log_WM.fbLogWM.M_Write_Log('FB_01_Action_PickToolMagazine : 2_AboveLocation=Error');
							PRG_Log_WM.fbLogWM.M_Write_Log(CONCAT('FB_01_Action_PickToolMagazine : ErrorID=',UDINT_TO_STRING(udiErrorID)));
						iSubStep:=0; // Stop SubStep
						iStep:=0; // Idle Step
					END_IF

				8: (* Start Y move *)
					GV_Axes.stAxisY.lrAutoPosAbs:=stToolLocation.lrYcoord;
					GV_Axes.stAxisY.bAutoCmdAbs:=TRUE;
					(*Log*)
						PRG_Log_WM.fbLogWM.M_Write_Log('FB_01_Action_PickToolMagazine : 2_AboveLocation : 8 : Start Y move');
					iSubStep:=9; // Next Step

				9: (* Wait Y move done *)
				   IF GV_Axes.stAxisY.bAutoDone AND (NOT bYError) THEN
						GV_Axes.stAxisY.bAutoCmdAbs:=FALSE;
						tonTimeoutMove2.IN:=FALSE;
						(*Log*)
							PRG_Log_WM.fbLogWM.M_Write_Log('FB_01_Action_PickToolMagazine : 2_AboveLocation : 9 : Y move done');
							PRG_Log_WM.fbLogWM.M_Write_Log('FB_01_Action_PickToolMagazine : 2_AboveLocation->3_GripperUnclamp');
						iSubStep:=0; // End SubStep
						iStep:=3; // Next Step
					ELSIF bYError THEN
						bError:=TRUE;
						udiErrorID:=291; // 291 = Step 2 SubStep 9 Error Axis Y 1
						GV_Axes.stAxisY.bAutoCmdAbs:=FALSE;
						tonTimeoutMove2.IN:=FALSE;
						(*Log*)
							PRG_Log_WM.fbLogWM.M_Write_Log('FB_01_Action_PickToolMagazine : 2_AboveLocation=Error');
							PRG_Log_WM.fbLogWM.M_Write_Log(CONCAT('FB_01_Action_PickToolMagazine : ErrorID=',UDINT_TO_STRING(udiErrorID)));
						iSubStep:=0; // Stop SubStep
						iStep:=0; // Idle Step
					END_IF
					
			END_CASE	
		
			IF tonTimeoutMove2.Q AND tonTimeoutMove2.PT<>T#0S THEN // Timeout 
				bError:=TRUE;
				udiErrorID:=299; // 299 = Step 2 Error Timeout 99
				GV_Axes.stAxisX.bAutoCmdAbs:=FALSE;
				GV_Axes.stAxisY.bAutoCmdAbs:=FALSE;
				GV_Axes.stAxisZ.bAutoCmdAbs:=FALSE;
				tonTimeoutMove2.IN:=FALSE;
				(*Log*)
					PRG_Log_WM.fbLogWM.M_Write_Log('FB_01_Action_PickToolMagazine : 2_AboveLocation=Error');
					PRG_Log_WM.fbLogWM.M_Write_Log(CONCAT('FB_01_Action_PickToolMagazine : ErrorID=',UDINT_TO_STRING(udiErrorID)));
				iSubStep:=0;
				iStep:=0;
			END_IF

		3: (* Step 3 = Operate manipulator gripper to unclamp *)
			eGripperMode:=ENUM_Gripper_Mode.Open; // Gripper mode
			tGripperTime:=tMouvementGripperOpen; // Gripper mouvement time
			bGripperSensor:=bCheckSensorGripperOpen; // Gripper check sensor
			
			IF (NOT fbGripper.bStart) AND (NOT fbGripper.bInit) AND (NOT fbGripper.bBusy) THEN // Gripper Start
				fbGripper.bStart:=TRUE;
			END_IF
			IF fbGripper.bDone AND (NOT fbGripper.bError) THEN // Gripper Done
				fbGripper.bStart:=FALSE;
				(*Log*)
					PRG_Log_WM.fbLogWM.M_Write_Log('FB_01_Action_PickToolMagazine : 3_GripperUnclamp->4_Location');
				iStep:=4; // Next Step
			ELSIF fbGripper.bError THEN // Gripper Error
				bError:=TRUE;
				udiErrorID:=300+fbGripper.udiErrorID; // 3xx = Step 3 Error + Error xx fbGripper
				fbGripper.bStart:=FALSE;
				(*Log*)
					PRG_Log_WM.fbLogWM.M_Write_Log('FB_01_Action_PickToolMagazine : 3_GripperUnclamp=Error');
					PRG_Log_WM.fbLogWM.M_Write_Log(CONCAT('FB_01_Action_PickToolMagazine : ErrorID=',UDINT_TO_STRING(udiErrorID)));
				iStep:=0; // Idle Step
			END_IF
		
		4: (* Step 4 = Move the manipulator on the tool/location (Z-1mm) *)
			tonTimeoutMove4.PT:=tMove4Timeout;
			tonTimeoutMove4.IN:=TRUE;
			
			CASE iSubStep OF
        
				0: (* Start Z-1 move *)
					GV_Axes.stAxisZ.lrAutoPosAbs:=stToolLocation.lrZcoord-1;
					GV_Axes.stAxisZ.bAutoCmdAbs:=TRUE;
					(*Log*)
						PRG_Log_WM.fbLogWM.M_Write_Log('FB_01_Action_PickToolMagazine : 4_Location : 0 : Start Z-1mm move');
					iSubStep:=1; // Next SubStep

				1: (* Wait Z-1 move done *)
				   IF GV_Axes.stAxisZ.bAutoDone AND (NOT bZError) THEN
						GV_Axes.stAxisZ.bAutoCmdAbs:=FALSE;
						tonTimeoutMove4.IN:=FALSE;
						(*Log*)
							PRG_Log_WM.fbLogWM.M_Write_Log('FB_01_Action_PickToolMagazine : 4_Location : 1 : Z-1mm move done');
							PRG_Log_WM.fbLogWM.M_Write_Log('FB_01_Action_PickToolMagazine : 4_Location->5_GripperClamp');
						iSubStep:=0; // End SubStep
						iStep:=5; // Next Step
					ELSIF bZError THEN
						bError:=TRUE;
						udiErrorID:=411; // 411 = Step 4 SubStep 1 Error Axis Z 1
						GV_Axes.stAxisZ.bAutoCmdAbs:=FALSE;
						tonTimeoutMove4.IN:=FALSE;
						(*Log*)
							PRG_Log_WM.fbLogWM.M_Write_Log('FB_01_Action_PickToolMagazine : 4_Location=Error');
							PRG_Log_WM.fbLogWM.M_Write_Log(CONCAT('FB_01_Action_PickToolMagazine : ErrorID=',UDINT_TO_STRING(udiErrorID)));
						iSubStep:=0; // Stop SubStep
						iStep:=0; // Idle Step
					END_IF
					
			END_CASE	
		
			IF tonTimeoutMove4.Q AND tonTimeoutMove4.PT<>T#0S THEN // Timeout 
				bError:=TRUE;
				udiErrorID:=499; // 499 = Step 4 Error Timeout 99
				GV_Axes.stAxisX.bAutoCmdAbs:=FALSE;
				GV_Axes.stAxisY.bAutoCmdAbs:=FALSE;
				GV_Axes.stAxisZ.bAutoCmdAbs:=FALSE;
				tonTimeoutMove4.IN := FALSE;
				(*Log*)
					PRG_Log_WM.fbLogWM.M_Write_Log('FB_01_Action_PickToolMagazine : 4_Location=Error');
					PRG_Log_WM.fbLogWM.M_Write_Log(CONCAT('FB_01_Action_PickToolMagazine : ErrorID=',UDINT_TO_STRING(udiErrorID)));
				iSubStep:=0;
				iStep:=0;
			END_IF

		5: (* Step 5 = Release manipulator gripper to clamp *)
			eGripperMode:=ENUM_Gripper_Mode.Close;
			tGripperTime:=tMouvementGripperClose; // Gripper mouvement time
			bGripperSensor:=bCheckSensorGripperClose; // Gripper check sensor
			
			IF (NOT fbGripper.bStart) AND (NOT fbGripper.bInit) AND (NOT fbGripper.bBusy) THEN // Gripper Start
				fbGripper.bStart:=TRUE;
			END_IF
			IF fbGripper.bDone AND (NOT fbGripper.bError) THEN // Gripper Done
				fbGripper.bStart:=FALSE;
				(*Memory*)
					//stToolLocation.bToolPresence:=FALSE; // Transfer Memory from Magazine to Manipulator
					IF stToolLocation.iAbsLocationNumber>0 AND stToolLocation.iAbsLocationNumber<=GV_Tool_Magazine.iMaxAbsLocation THEN
						GV_Tool_Magazine.aLocation[stToolLocation.iAbsLocationNumber].bToolPresence:=FALSE; // Transfer Memory from Magazine to Manipulator
					END_IF
					GV_Tool_Magazine.stManipulator.iAbsLocationNumberMemory:=stToolLocation.iAbsLocationNumber; // Transfer Memory from Magazine to Manipulator
					GV_Tool_Magazine.stManipulator.iRelLocationNumberMemory:=stToolLocation.iRelLocationNumber; // Transfer Memory from Magazine to Manipulator
					
				(*Log*)
					PRG_Log_WM.fbLogWM.M_Write_Log('FB_01_Action_PickToolMagazine : 5_GripperClamp->6_FrontLocation');
				iStep:=6; // Next Step
			ELSIF fbGripper.bError THEN // Gripper Error
				bBusy:=FALSE;
				bError:=TRUE;
				udiErrorID:=500+fbGripper.udiErrorID; // 5xx = Step 5 Error + Error xx fbGripper
				fbGripper.bStart:=FALSE;
				(*Log*)
					PRG_Log_WM.fbLogWM.M_Write_Log('FB_01_Action_PickToolMagazine : 5_GripperClamp=Error');
					PRG_Log_WM.fbLogWM.M_Write_Log(CONCAT('FB_01_Action_PickToolMagazine : ErrorID=',UDINT_TO_STRING(udiErrorID)));
				iStep:=0; // Idle Step
			END_IF
		
		6: (* Step 6 = Move the manipulator in front of tool/location (Z->YHome) -> Pull the tool from the magazine *)
			tonTimeoutMove6.PT:=tMove6Timeout;
			tonTimeoutMove6.IN:=TRUE;
			
			CASE iSubStep OF
        
				0: (* Start Z move *)
					GV_Axes.stAxisZ.lrAutoPosAbs:=stToolLocation.lrZcoord;
					GV_Axes.stAxisZ.bAutoCmdAbs:=TRUE;
					(*Log*)
						PRG_Log_WM.fbLogWM.M_Write_Log('FB_01_Action_PickToolMagazine : 6_FrontLocation : 0 : Start Z');
					iSubStep:=1; // Next SubStep

				1: (* Wait Z move done *)
				   IF GV_Axes.stAxisZ.bAutoDone AND (NOT bZError) THEN
						GV_Axes.stAxisZ.bAutoCmdAbs:=FALSE;
						(*Log*)
							PRG_Log_WM.fbLogWM.M_Write_Log('FB_01_Action_PickToolMagazine : 6_FrontLocation : 1 : Z move done');
						iSubStep:=2; // Next SubStep
					ELSIF bZError THEN
						bError:=TRUE;
						udiErrorID:=611; // 611 = Step 6 SubStep 1 Error Axis Z 1
						GV_Axes.stAxisZ.bAutoCmdAbs:=FALSE;
						tonTimeoutMove6.IN:=FALSE;
						(*Log*)
							PRG_Log_WM.fbLogWM.M_Write_Log('FB_01_Action_PickToolMagazine : 6_FrontLocation=Error');
							PRG_Log_WM.fbLogWM.M_Write_Log(CONCAT('FB_01_Action_PickToolMagazine : ErrorID=',UDINT_TO_STRING(udiErrorID)));
						iSubStep:=0; // Stop SubStep
						iStep:=0; // Idle Step
					END_IF
		
				2: (* Start YHome move *)
					GV_Axes.stAxisY.lrAutoPosAbs:=GV_Tool_Magazine.stManipulator.lrYHome;
					GV_Axes.stAxisY.bAutoCmdAbs:=TRUE;
					(*Log*)
						PRG_Log_WM.fbLogWM.M_Write_Log('FB_01_Action_PickToolMagazine : 6_FrontLocation : 2 : Start YHome move');
					iSubStep:=3; // Next SubStep

				3: (* Wait YHome move done *)
				   IF GV_Axes.stAxisY.bAutoDone AND (NOT bYError) THEN
						GV_Axes.stAxisY.bAutoCmdAbs:=FALSE;
						tonTimeoutMove6.IN:=FALSE;
						(*Log*)
							PRG_Log_WM.fbLogWM.M_Write_Log('FB_01_Action_PickToolMagazine : 6_FrontLocation : 3 : YHome move done');
							PRG_Log_WM.fbLogWM.M_Write_Log('FB_01_Action_PickToolMagazine : 6_FrontLocation->7_Tunnel');
						iSubStep:=0; // End SubStep
						iStep:=7; // Next Step
					ELSIF bYError THEN
						bError:=TRUE;
						udiErrorID:=631; // 631 = Step 6 SubStep 3 Error Axis Y 1
						GV_Axes.stAxisY.bAutoCmdAbs:=FALSE;
						tonTimeoutMove6.IN:=FALSE;
						(*Log*)
							PRG_Log_WM.fbLogWM.M_Write_Log('FB_01_Action_PickToolMagazine : 6_FrontLocation=Error');
							PRG_Log_WM.fbLogWM.M_Write_Log(CONCAT('FB_01_Action_PickToolMagazine : ErrorID=',UDINT_TO_STRING(udiErrorID)));
						iSubStep:=0; // Stop SubStep
						iStep:=0; // Idle Step
					END_IF
					
			END_CASE	
		
			IF tonTimeoutMove6.Q AND tonTimeoutMove6.PT<>T#0S THEN // Timeout 
				bError:=TRUE;
				udiErrorID:=699; // 699 = Step 6 Error Timeout 99
				GV_Axes.stAxisX.bAutoCmdAbs:=FALSE;
				GV_Axes.stAxisY.bAutoCmdAbs:=FALSE;
				GV_Axes.stAxisZ.bAutoCmdAbs:=FALSE;
				tonTimeoutMove6.IN := FALSE;
				(*Log*)
					PRG_Log_WM.fbLogWM.M_Write_Log('FB_01_Action_PickToolMagazine : 6_FrontLocation=Error');
					PRG_Log_WM.fbLogWM.M_Write_Log(CONCAT('FB_01_Action_PickToolMagazine : ErrorID=',UDINT_TO_STRING(udiErrorID)));
				iSubStep:=0;
				iStep:=0;
			END_IF
		
		7: (* Step 7 = Tunnel passage (if needed) *)
			IF (NOT bTunnelTravel) THEN
				IF GV_Tool_Magazine.stManipulator.ePositionMag=ENUM_Position_Magazine.Top THEN
					bTunnelTravel:=FALSE;
					(*Log*)
						PRG_Log_WM.fbLogWM.M_Write_Log('FB_01_Action_PickToolMagazine : 7_Tunnel->0_Idle');
						//PRG_Log_WM.fbLogWM.M_Write_Log('FB_01_Action_PickToolMagazine : 7_Tunnel->8_PositionTransferArm');
					iSubStep:=0; // End SubStep
					iStep:=0; // Idle Step
					bDone:=TRUE;
					bBusy:=FALSE;
					 //iStep:=8; // Next Step
				END_IF	
				IF GV_Tool_Magazine.stManipulator.ePositionMag=ENUM_Position_Magazine.Bottom THEN
					eTunnelMode:=ENUM_Tunnel_MODE.BottomToTop;
					bTunnelTravel:=TRUE;
					(*Log*)
						PRG_Log_WM.fbLogWM.M_Write_Log('FB_01_Action_PickToolMagazine : 7_Tunnel : Need to Travel Bottom->Top');
				END_IF			
				IF GV_Tool_Magazine.stManipulator.ePositionMag=ENUM_Position_Magazine.Unknow THEN // Manipulator Unknow position
					bError:=TRUE;
					udiErrorID:=701; // 701 = Step 7 Error Tunnel 01
					fbTunnel.bStart:=FALSE;
					bTunnelTravel:=FALSE;
					(*Log*)
						PRG_Log_WM.fbLogWM.M_Write_Log('FB_01_Action_PickToolMagazine : 7_Tunnel=Error');
						PRG_Log_WM.fbLogWM.M_Write_Log(CONCAT('FB_01_Action_PickToolMagazine : ErrorID=',UDINT_TO_STRING(udiErrorID)));
					iStep:=0; // Idle Step
				END_IF
			END_IF
			
			IF bTunnelTravel AND (NOT fbTunnel.bStart) AND (NOT fbTunnel.bInit) AND (NOT fbTunnel.bBusy) THEN // Tunnel Start
				fbTunnel.bStart:=TRUE;
			END_IF
			IF fbTunnel.bDone AND (NOT fbTunnel.bError) THEN // Tunnel Done
				fbTunnel.bStart:=FALSE;
				bTunnelTravel:=FALSE;
				(*Log*)
					PRG_Log_WM.fbLogWM.M_Write_Log('FB_01_Action_PickToolMagazine : 7_Tunnel->0_Idle');
					//PRG_Log_WM.fbLogWM.M_Write_Log('FB_01_Action_PickToolMagazine : 7_Tunnel->8_PositionTransferArm');
				iSubStep:=0; // End SubStep
				iStep:=0; // Idle Step
				bDone:=TRUE;
				bBusy:=FALSE;
				//iStep:=8; // Next Step
			ELSIF fbTunnel.bError THEN // Tunnel Error
				bError:=TRUE;
				udiErrorID:=700+fbTunnel.udiErrorID; // 7xx = Step 7 Error + Error xx fbTunnel
				fbTunnel.bStart:=FALSE;
				bTunnelTravel:=FALSE;
				(*Log*)
					PRG_Log_WM.fbLogWM.M_Write_Log('FB_01_Action_PickToolMagazine : 7_Tunnel=Error');
					PRG_Log_WM.fbLogWM.M_Write_Log(CONCAT('FB_01_Action_PickToolMagazine : ErrorID=',UDINT_TO_STRING(udiErrorID)));
				iStep:=0; // Idle Step
			END_IF
			
// 		8: (* Step 8 = Move the manipulator to be ready for the transfer to the Changing Arm (X->Z) *)
// 			tonTimeoutMove8.PT:=tMove8Timeout;
// 			tonTimeoutMove8.IN:=TRUE;
// 			
// 			CASE iSubStep OF
//         
// 				0: (* Start ZLowestRackTop move *)
// 					GV_Axes.stAxisZ.lrAutoPosAbs:=GV_Tool_Magazine.lrZLowestRackTop+40;//GV_Tool_Magazine.stManipulator.lrZTunnelTop;
// 					GV_Axes.stAxisZ.bAutoCmdAbs:=TRUE;
// 					(*Log*)
// 						PRG_Log_WM.fbLogWM.M_Write_Log('FB_01_Action_PickToolMagazine : 8_PositionTransferArm : 0 : Start ZLowestRackTop move');
// 					iSubStep:=1; // Next SubStep
// 					
// 				1: (* Wait ZLowestRackTop move done *)
// 				   IF GV_Axes.stAxisZ.bAutoDone AND (NOT bZError) THEN
// 						GV_Axes.stAxisZ.bAutoCmdAbs:=FALSE;
// 						(*Log*)
// 							PRG_Log_WM.fbLogWM.M_Write_Log('FB_01_Action_PickToolMagazine : 8_PositionTransferArm : 0 : ZLowestRackTop move done');
// 						iSubStep:=2; // Next SubStep
// 					ELSIF bZError THEN
// 						bError:=TRUE;
// 						udiErrorID:=811; // 811 = Step 8 SubStep 1 Error Axis Z 1
// 						GV_Axes.stAxisZ.bAutoCmdAbs:=FALSE;
// 						tonTimeoutMove2.IN:=FALSE;
// 						(*Log*)
// 							PRG_Log_WM.fbLogWM.M_Write_Log('FB_01_Action_PickToolMagazine : 8_PositionTransferArm=Error');
// 							PRG_Log_WM.fbLogWM.M_Write_Log(CONCAT('FB_01_Action_PickToolMagazine : ErrorID=',UDINT_TO_STRING(udiErrorID)));
// 						iSubStep:=0; // Stop SubStep
// 						iStep:=0; // Idle Step
// 					END_IF
// 		
// 				2: (* Start X move *)
// 					GV_Axes.stAxisX.lrAutoPosAbs:=GV_Axes.stAxisX.lrAutoPosAbs:=GV_Tool_Magazine.stManipulator.lrXTransferGripper1;
// 					GV_Axes.stAxisX.bAutoCmdAbs:=TRUE;
// 					(*Log*)
// 						PRG_Log_WM.fbLogWM.M_Write_Log('FB_01_Action_PickToolMagazine : 8_PositionTransferArm : 2 : Start X move');
// 					iSubStep:=3; // Next SubStep
// 
// 				3: (* Wait X move done *)
// 				   IF GV_Axes.stAxisX.bAutoDone AND (NOT bXError) THEN
// 						GV_Axes.stAxisX.bAutoCmdAbs:=FALSE;
// 						(*Log*)
// 							PRG_Log_WM.fbLogWM.M_Write_Log('FB_01_Action_PickToolMagazine : 8_PositionTransferArm : 3 : X move done');
// 						iSubStep:=0; // End SubStep
// 						iStep:=0; // Idle Step
// 						bDone:=TRUE;
// 						bBusy:=FALSE;
// 					ELSIF bXError THEN
// 						bError:=TRUE;
// 						udiErrorID:=831; // 831 = Step 8 SubStep 3 Error Axis X 1
// 						GV_Axes.stAxisX.bAutoCmdAbs:=FALSE;
// 						tonTimeoutMove8.IN:=FALSE;
// 						(*Log*)
// 							PRG_Log_WM.fbLogWM.M_Write_Log('FB_01_Action_PickToolMagazine : 8_PositionTransferArm=Error');
// 							PRG_Log_WM.fbLogWM.M_Write_Log(CONCAT('FB_01_Action_PickToolMagazine : ErrorID=',UDINT_TO_STRING(udiErrorID)));
// 						iSubStep:=0; // Stop SubStep
// 						iStep:=0; // Idle Step
// 					END_IF
// 					
// 			END_CASE	
// 		
// 			IF tonTimeoutMove8.Q AND tonTimeoutMove8.PT<>T#0S THEN // Timeout 
// 				bError:=TRUE;
// 				udiErrorID:=899; // 899 = Step 8 Error Timeout 99
// 				GV_Axes.stAxisX.bAutoCmdAbs:=FALSE;
// 				GV_Axes.stAxisY.bAutoCmdAbs:=FALSE;
// 				GV_Axes.stAxisZ.bAutoCmdAbs:=FALSE;
// 				tonTimeoutMove8.IN := FALSE;
// 				(*Log*)
// 					PRG_Log_WM.fbLogWM.M_Write_Log('FB_01_Action_PickToolMagazine : 8_PositionTransferArm=Error');
// 					PRG_Log_WM.fbLogWM.M_Write_Log(CONCAT('FB_01_Action_PickToolMagazine : ErrorID=',UDINT_TO_STRING(udiErrorID)));
// 				iSubStep:=0;
// 				iStep:=0;
// 			END_IF		

	END_CASE

END_FUNCTION_BLOCK

// ---- 09_Tool_Magazine/03_POUs/02_FBs/FB_Manipulator_Gripper.TcPOU
FUNCTION_BLOCK FB_Manipulator_Gripper
VAR_INPUT
	(** SETUP ENUM **)
		eGripperMode : ENUM_Gripper_Mode ; // Mode of the gripper	

	(** SETUP TIME **)
		tMouvementDuration : TIME ; // Duration of the mouvement

	(** SETUP FLAG **)
		bSensorCheck : BOOL ; // With or without check of the presence sensor

	(** PROCESS FLAG **)
		bInit : BOOL ; // Init the FB
	    bStart : BOOL ; // Start the Fb
END_VAR
VAR_OUTPUT
	(** PROCESS UDINT **)
		udiErrorID : UDINT ; // Fb Error ID
		
	(** PROCESS FLAG **)
		bBusy  : BOOL ; // Fb is Busy
		bDone  : BOOL ; // Fb is Done
		bError : BOOL ; // Fb in Error
END_VAR
VAR_IN_OUT
END_VAR	
VAR
	(** STRING **)
		strTextLog : STRING ; // Text to Log

	(** PROCESS INT **)
		iStep  : INT := 0 ; // Step of the Fb
		iSubStep : INT := 0 ; // SubStep of the Fb
		iPrevStep : INT := 0 ; // Previous Step of the Fb
		iPrevSubStep : INT := 0 ; // Previous Subtep of the Fb
	
	(** PROCESS FLAG + R_TRIG **)
		rtInit : R_TRIG ; // FB Init at rising edge
		rtStart : R_TRIG ; // FB Start at rising edge
	
	(** FB **)
		tonWaitMouvement : TON ; // TON to wait the mouvement duration before the check
END_VAR

//-----------------------------------------------------------------------------------------
//
//                  			FB_Manipulator_Gripper
//
//				Motion control of the BERG gripper of the manipulator
//-----------------------------------------------------------------------------------------
//
//Auteur: G.GOETZ
//Création: 05.02.2026
//Dernière modification : 08.04.2026 (G.GOETZ)
//       			
//-----------------------------------------------------------------------------------------
//
//     							Liste des modifications  	
//
// 05.02.2026 (G.GOETZ) -> Création
// 08.04.2026 (G.GOETZ) -> Ajout Init
//-----------------------------------------------------------------------------------------

(** FB CALL **)
	rtInit(CLK:=bInit);
	rtStart(CLK:=bStart);
	
	tonWaitMouvement();

(** INIT **)
	IF (rtinit.Q OR bInit) AND (NOT bStart) THEN
		iStep:=0;
		bInit:=FALSE;
	END_IF

(** STEPS **)
    CASE iStep OF
		
        0: (* Step 0 = Idle *)
            bBusy:=FALSE;
            bDone:=FALSE;
			bError:=FALSE;
			udiErrorID:=0;
			iSubStep:=0;
			
			tonWaitMouvement.IN:=FALSE;
			
			(* Idle->Setup *)
				IF bStart AND (NOT bInit) THEN
					bBusy:=TRUE;
					(*Log*)
						PRG_Log_WM.fbLogWM.M_Write_Log('FB_Manipulator_Gripper : 0_Idle->1_Setup');
					iStep:=1; // Next Step
				END_IF
				
		1: (* Step 1 = Setup *)
			(*Log*)
				(*GripperMode*)
					CASE eGripperMode OF
						ENUM_Gripper_Mode.Open:		strTextLog:='Open';
						ENUM_Gripper_Mode.Close:	strTextLog:='Close';
					END_CASE
					PRG_Log_WM.fbLogWM.M_Write_Log(CONCAT('FB_Manipulator_Gripper : 1_Setup : Gripper Mode = ',strTextLog));
				(*SensorCheck*)
					IF bSensorCheck THEN
						strTextLog:='With';
					ELSE
						strTextLog:='Without';
					END_IF
					PRG_Log_WM.fbLogWM.M_Write_Log(CONCAT('FB_Manipulator_Gripper : 1_Setup : Sensor Check = ',strTextLog));
				(*MouvementDuration*)
					strTextLog:=TIME_TO_STRING(tMouvementDuration);
					PRG_Log_WM.fbLogWM.M_Write_Log(CONCAT('FB_Manipulator_Gripper : 1_Setup : Mouvement Duration = ',strTextLog));				
				PRG_Log_WM.fbLogWM.M_Write_Log('FB_Manipulator_Gripper : 1_Setup->2_Process');
				
			tonWaitMouvement.PT:=tMouvementDuration;
			iStep:=2; // Next Step
			
		2: (* Step 2 = Process *)
			tonWaitMouvement.IN:=TRUE; // Start TON mouvement
			
			CASE eGripperMode OF 
				
				ENUM_Gripper_Mode.Open: // Open = Unclamp
					GV_CNC.stFanucData.stMagazineCNC.boOpenManipulatorGripper:=TRUE; // Ask to the CNC to Open the Gripper
					IF tonWaitMouvement.Q THEN
						IF bSensorCheck THEN // With Sensor Check
							IF (NOT GV_IO.diToolPresenceCone) THEN // Sensor
								(*Log*)
									PRG_Log_WM.fbLogWM.M_Write_Log('FB_Manipulator_Gripper : 2_Process : Done with success');
									PRG_Log_WM.fbLogWM.M_Write_Log('FB_Manipulator_Gripper : 2_Process->0_Idle');
								iStep:=0; // Idle Step
								bDone:=TRUE;
								bBusy:=FALSE;
							ELSE
								bError:=TRUE;
								udiErrorID:=21; // 21 = Step 2 Error 1
								(*Log*)
									PRG_Log_WM.fbLogWM.M_Write_Log('FB_Manipulator_Gripper : 2_Process :Error');
									PRG_Log_WM.fbLogWM.M_Write_Log(CONCAT('FB_Manipulator_Gripper : ErrorID = ',UDINT_TO_STRING(udiErrorID)));
								iStep:=0; // Idle Step
							END_IF
						ELSE // Without Sensor Check
							(*Log*)
								PRG_Log_WM.fbLogWM.M_Write_Log('FB_Manipulator_Gripper : 2_Process : Done with success');
								PRG_Log_WM.fbLogWM.M_Write_Log('FB_Manipulator_Gripper : 2_Process->0_Idle');
							iStep:=0; // Idle Step
							bDone:=TRUE;
							bBusy:=FALSE;
						END_IF
					END_IF
		
				ENUM_Gripper_Mode.Close: // Close = Clamp
					GV_CNC.stFanucData.stMagazineCNC.boOpenManipulatorGripper:=FALSE; // Ask to the CNC to Closen the Gripper
					IF tonWaitMouvement.Q THEN
						IF bSensorCheck THEN // With Sensor Check
							IF GV_IO.diToolPresenceCone THEN // Sensor
								(*Log*)
									PRG_Log_WM.fbLogWM.M_Write_Log('FB_Manipulator_Gripper : 2_Process : Done with success');
									PRG_Log_WM.fbLogWM.M_Write_Log('FB_Manipulator_Gripper : 2_Process->0_Idle');
								iStep:=0; // Idle Step
								bDone:=TRUE;
								bBusy:=FALSE;
							ELSE
								bError:=TRUE;
								udiErrorID:=22; // 22 = Step 2 Error 2
								(*Log*)
									PRG_Log_WM.fbLogWM.M_Write_Log('FB_Manipulator_Gripper : 2_Process :Error');
									PRG_Log_WM.fbLogWM.M_Write_Log(CONCAT('FB_Manipulator_Gripper : ErrorID = ',UDINT_TO_STRING(udiErrorID)));
								iStep:=0; // Idle Step
							END_IF
						ELSE // Without Sensor Check
							(*Log*)
								PRG_Log_WM.fbLogWM.M_Write_Log('FB_Manipulator_Gripper : 2_Process : Done with success');
								PRG_Log_WM.fbLogWM.M_Write_Log('FB_Manipulator_Gripper : 2_Process->0_Idle');
							iStep:=0; // Idle Step
							bDone:=TRUE;
							bBusy:=FALSE;
						END_IF
					END_IF
					
			END_CASE
			
	END_CASE

END_FUNCTION_BLOCK

// ---- 08_Cycle/03_POUs/02_FBs/FB_02_Action_TransferManipulatorToArm.TcPOU
FUNCTION_BLOCK FB_02_Action_TransferManipulatorToArm
VAR_INPUT
	(** SETUP ST **)
		//stToolLocation : ST_Tool_Location ; // Tool_Location structure of the Tool to Transfer
		
	(** SETUP TIME **)
		(*Manipulator Gripper mvmnt*)
			tMouvementGripperOpen : TIME ; // Value of the manipulator gripper open mouvement duration
			tMouvementGripperClose : TIME ; // Value of the manipulator gripper close mouvement duration
		(*Tunnel*)
			tTunnelTimeout : TIME ; // Value of the timeout for travel the tunnel
		(*Step 2*)
			tMove2Timeout : TIME ; // Value of the timeout for Step 2
		(*Step 3*)
			tMove3Timeout : TIME ; // Value of the timeout for Step 3
		(*Step 4*)
			tMove4Timeout : TIME ; // Value of the timeout for Step 4
		(*Step 5*)
			tMove5Timeout : TIME ; // Value of the timeout for Step 5
		(*Step 7*)
			tMove7Timeout : TIME ; // Value of the timeout for Step 7
	
	(** SETUP REAL **)

	(** SETUP INT **)
		iGripperArmNumber : INT ; // Arm gripper number for the transfer
	
	(** SETUP FLAG **)
		bCheckSensorManipulatorGripper : BOOL ; // Check the manipulator gripper sensor at the beginning
		bCheckSensorArmGripper1 : BOOL ; // Check the arm gripper 1 sensor at the beginning
		bCheckSensorArmGripper2 : BOOL ; // Check the arm gripper 2 sensor at the beginning
		(*Gripper*)
			bCheckSensorGripperOpen : BOOL ; // Check the manipulator gripper sensor after open
			bCheckSensorGripperClose : BOOL ; // Check the manipulator gripper sensor after close	
			
	(** PROCESS FLAG **)
		bInit : BOOL ;  // Init the Fb
	    bStart : BOOL ; // Start the Fb
END_VAR
VAR_OUTPUT
	(** PROCESS UDINT **)
		udiErrorID : UDINT ; // Fb Error ID
		
	(** PROCESS FLAG **)
		bBusy  : BOOL ; // Fb is Busy
		bDone  : BOOL ; // Fb is Done
		bError : BOOL ; // Fb in Error
END_VAR
VAR_IN_OUT
END_VAR	
VAR
	(** SETUP ENUM **)
		(*Manipulator Gripper mvmnt*)
			eGripperMode : ENUM_Gripper_Mode; // Gripper mode for gripper mouvement (fbGripper)
		(*Tunnel*)
			eTunnelMode : ENUM_Tunnel_Mode; // Tunnel mode for travel (fbTunnel)

	(** SETUP TIME **)
		(*Manipulator Gripper mvmnt*)
			tGripperTime : TIME ; // Mouvement duration for gripper mouvement (fbGripper)
	
	(** SETUP FLAG **)
		(*Manipulator Gripper mvmnt*)
			bGripperSensor : BOOL ; // Sensor check for gripper mouvement (fbGripper)
		
	(** PROCESS STRING **)
		strTextLog : STRING ; // Text to Log
		
	(** PROCESS INT **)
		iStep  : INT := 0 ; // Step of the Fb
		iSubStep : INT := 0 ; // SubStep of the Fb
		iPrevStep : INT := 0 ; // Previous Step of the Fb
		iPrevSubStep : INT := 0 ; // Previous Subtep of the Fb
			
	(** PROCESS FLAG + R_TRIG **)
		rtInit : R_TRIG ; // FB Init at rising edge
		rtStart : R_TRIG ; // FB Start at rising edge
		(*Tunnel*)
			bTunnelTravel : BOOL ; // Need to travel the tunnel
		bXError : BOOL ; // Axis X Error
		bYError : BOOL ; // Axis Y Error
		bZError : BOOL ; // Axis Z Error
		bArmError : BOOL ; // Axis Arm Error
		
		
	(** FB **)
		(*Gripper*)
			fbGripper : FB_Manipulator_Gripper ;
		(*Tunnel*)
			fbTunnel : FB_Manipulator_Tunnel ;
		(*Step 2*)
			tonTimeoutMove2 : TON ; // TON timeout for the Step 2
		(*Step 3*)
			tonTimeoutMove3 : TON ; // TON timeout for the Step 3
		(*Step 4*)
			tonTimeoutMove4 : TON ; // TON timeout for the Step 4
		(*Step 5*)
			tonTimeoutMove5 : TON ; // TON timeout for the Step 5
		(*Step 7*)
			tonTimeoutMove7 : TON ; // TON timeout for the Step 7
END_VAR

//-----------------------------------------------------------------------------------------
//
//                  		FB_02_Action_TransferManipulatorToArm
//
//		Management of the tool transfer from the Manipulator to the Changing arm
//-----------------------------------------------------------------------------------------
//
//Auteur: G.GOETZ
//Création: 09.02.2026
//Dernière modification : 09.02.2026 (G.GOETZ)
//       			
//-----------------------------------------------------------------------------------------
//
//     							Liste des modifications  	
//
// 09.02.2026 (G.GOETZ) -> Création
// 09.04.2026 (G.GOETZ) -> Ajout Init + Modification du cycle
//-----------------------------------------------------------------------------------------

(** FB CALL **)
	rtInit(CLK:=bInit);
	rtStart(CLK:=bStart);
	
